// TIA Portal V20 export
FUNCTION_BLOCK "CallEquipment"   // FB134, LAD
TITLE = CallEquipment
// This block includes all general functions, checks and logik that is needed in the entire unit. E.g. general releases and system wide functionalities like air, pressure and power handling as well as general reaction to events.
// stored: IsIECCheckEnabled true, MemoryReserve 100, Namespace Unit1.Em0, SetENOAutomatically true
   VAR_INPUT
      ZoneOperationEnable { ExternalWritable := 'False'} : "LWONIK_typeSafetyZoneManualOperation";
      unitEnableControlInterfaces { ExternalWritable := 'False'} : "LAF_typeEnableControlInterfaces";
      commandExcute { ExternalWritable := 'False'} : Bool;
   END_VAR
   VAR_IN_OUT
      unitStatus : "LAF_typeUnitStatus";   // Current unit status o be used in this EM
      emFeedback : "LUC_typeEmFeedback";   // Feedback of the EM to the Unit
      unitAlarmDB : "LAF_typeAlarms";   // Summarized EM Alarms for the Unit
   END_VAR
   VAR
      instSequenceUnWinder { ExternalWritable := 'False'} : "Unit1.Em0.Sequence_1_UnWinder";   // EM Sequence Instance
      instUnWinderInitializedJob1 { ExternalWritable := 'False'} : "LAF_SelectJob";
      instUnWinderRunJob2 { ExternalWritable := 'False'} : "LAF_SelectJob";
      instUnWinderStopJob3 { ExternalWritable := 'False'} : "LAF_SelectJob";
      instUnWinderRewindJob4 { ExternalWritable := 'False'} : "LAF_SelectJob";
      instCmUnWinderAxisB { ExternalWritable := 'False'} : "LBC_AxisControl_TecPlcCn";
      instCmAirShaftOnOff { ExternalWritable := 'False'} : "LBC_TwoWayActuatorCn";
      instcmExpelFwdBwd { ExternalWritable := 'False'} : "LBC_TwoWayActuatorCn";
      instCmTensionCheckSensor { ExternalWritable := 'False'} : "LBC_DigitalSignalCn";
      instCmRadiusMeasureAnalogInput { ExternalWritable := 'False'} : "LBC_AnalogInputCn";
      instCmEpc { ExternalWritable := 'False'} : "LER_EPC_CON600";
      instCmRadiusMeasure { ExternalWritable := 'False'} : "LER_RadiusMeasure";
      instUnWinderAxisControlInterlockSummary { ExternalWritable := 'False'} : "LER_AxisControl_InterlockSummary";
      instServoTorqueCal_DR1 { ExternalWritable := 'False'} : "LER_ServoTorqueCal";
      instLDrv701ControlUnWinderAxisB { ExternalWritable := 'False'} : "LDrvSafe_SinaTlg701Control";   // Drive Telegram Function Library
      instLDrv701StatusUnWinderAxisB { ExternalWritable := 'False'} : "LDrvSafe_SinaTlg701Status";   // Drive Telegram Function Library
      statUnitStatus { ExternalWritable := 'False'} : "LAF_typeUnitStatus";   // Unit Status that is used in this project
      statAllBrakeTest { ExternalWritable := 'False'} : "LER_typeBrakeTestUnitCommands";
      instManageAlarms { ExternalWritable := 'False'} : "LAF_ManageAlarms";
      instEventsPFE { S7_SetPoint := 'True'} : "Unit1.Em0.EventsPFE";
      statEnableManualCmds { ExternalWritable := 'False'} : Bool;
      statRcEnableCmds { ExternalWritable := 'False'} : Bool;
      statPulse { ExternalWritable := 'False'} : Array[0..99] of Bool;
      statTonTimer { ExternalWritable := 'False'} : Array[0..99] of TON_TIME;
      statTofTimer { ExternalWritable := 'False'} : Array[0..99] of TOF_TIME;
      statRadius { ExternalWritable := 'False'} : LReal;
      statDiameter { ExternalWritable := 'False'} : LReal;
      citi_Ptrig : Array[0..20] of Bool;
      citiTon : Array[0..20] of TON_TIME;
      citi : Time;
      citiTest : Array[0..20] of Bool;
      SpeedLimitByRadius_Instance { S7_SetPoint := 'True'} : "Unit1.Em0.SpeedLimitByRadius";
      SpeedLimit : LReal;
      SpeedRef : LReal;
      SinaParaS_Instance { S7_SetPoint := 'True'} : SinaParaS;
   END_VAR
   VAR_TEMP
      tempScInProduction : Bool;   // Mode Production and StateComplete
      tempScNoProduction : Bool;   // Mode Manual and StateComplete
   END_VAR
   VAR CONSTANT
      TO_DO_INSERT_PRECONDITIONS_HERE : Bool := TRUE;   // Template : Add em specific conditions here
      NO_JOB : DInt;   // No job
      TRUE : Bool := TRUE;
      FALSE : Bool := FALSE;
   END_VAR
   VAR_TEMP   // added for the SCL form of the ladder/FBD networks
      _w1 : Bool;
      _w2 : Bool;
      _w3 : Bool;
      _w4 : Bool;
      _w5 : Bool;
      _w6 : Bool;
      _w7 : Bool;
      _w8 : Bool;
      _w9 : Bool;
      _w10 : Bool;
      _w11 : Bool;
      _w12 : Bool;
      _w13 : Bool;
      _w14 : Bool;
      _w15 : Bool;
   END_VAR
BEGIN

REGION Network 1: BLOCK INFO HEADER
   // (company) / (C) Copyright (year)
   // ---------------------------------------------------------------------------------
   // Title:                             (Title of this block)
   // Comment/Function: (that is implemented in the block)
   // Library/Family:           (that the source is dedicated to)
   // Author:                        (department / person in charge / contact)
   // Target System:          (test system with FW version)
   // Engineering:              TIA Portal (SW version)
   // Restrictions:               (OB types, etc.)
   // Requirements:           (hardware, technological package, etc.)
   // ---------------------------------------------------------------------------------
   // Change log table:
   // Version          | Date             | Signature      | Expert in charge  | Changes applied ------------------------|----------------------|-------------------------|--------------------------------|-----------------------
   // 001.000.000 | yyyy-mm-dd | 0x00000000 | (name of expert) | First released version
END_REGION

REGION Network 2: DESCRIPTION
   // This is a template block provided by the Automation Framework. It can be used to create an own project.
   // The Block Info Header is prepared to put in your own data.
   // Description of the block could be added here and the docu created by Code2Docu.
END_REGION

REGION Network 3: ******************** Unit Input ********************
END_REGION

REGION Network 4: Em Nodes Brake Test
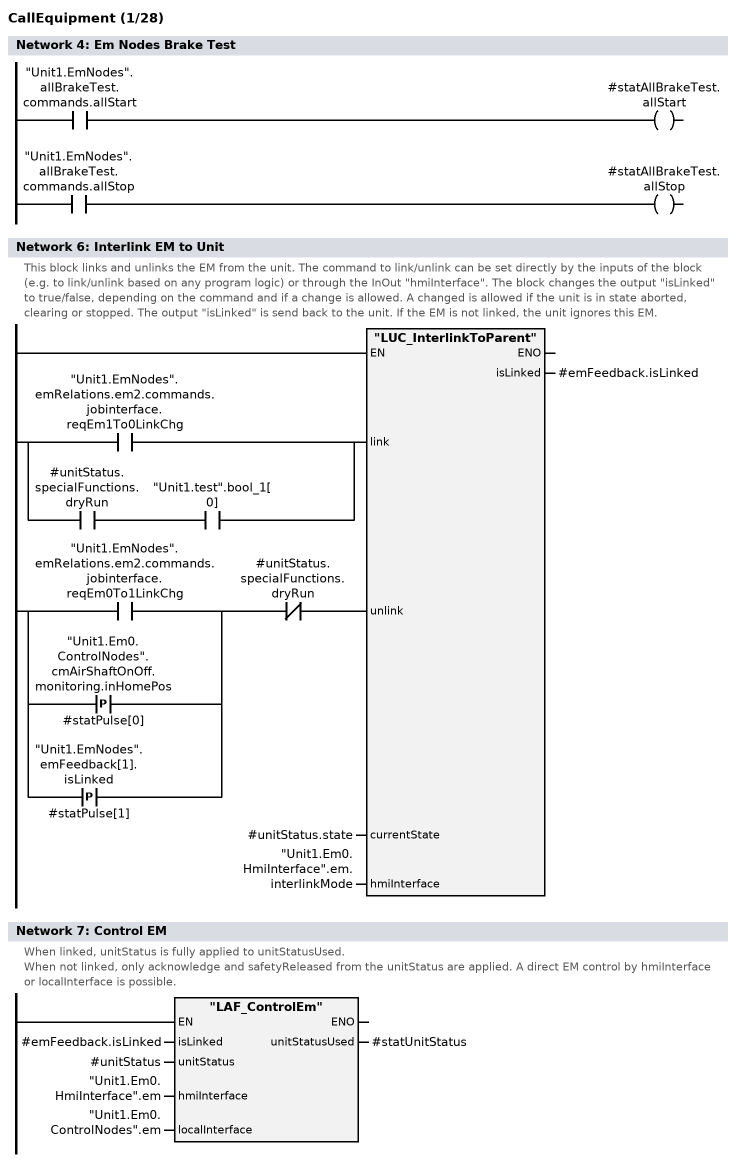
   RUNG wire#powerrail
      Contact( "Unit1.EmNodes".allBrakeTest.commands.allStart )
      Coil( #statAllBrakeTest.allStart )
   END_RUNG
   RUNG wire#powerrail
      Contact( "Unit1.EmNodes".allBrakeTest.commands.allStop )
      Coil( #statAllBrakeTest.allStop )
   END_RUNG
   // the same network as SCL:
   #statAllBrakeTest.allStart := "Unit1.EmNodes".allBrakeTest.commands.allStart;
   #statAllBrakeTest.allStop := "Unit1.EmNodes".allBrakeTest.commands.allStop;
END_REGION

REGION Network 5: ******************** Equipment Control ********************
END_REGION

REGION Network 6: Interlink EM to Unit
   // This block links and unlinks the EM from the unit. The command to link/unlink can be set directly by the inputs of the block (e.g. to link/unlink based on any program logic) or through the InOut "hmiInterface". The block changes the output "isLinked" to true/false, depending on the command and if a change is allowed. A changed is allowed if the unit is in state aborted, clearing or stopped. The output "isLinked" is send back to the unit. If the EM is not linked, the unit ignores this EM.
   RUNG wire#powerrail
      "LUC_InterlinkToParent"(link := wire#w1, unlink := wire#w3, currentState := #unitStatus.state, hmiInterface := "Unit1.Em0.HmiInterface".em.interlinkMode, isLinked => #emFeedback.isLinked)
   END_RUNG
   RUNG wire#powerrail
      Contact( "Unit1.EmNodes".emRelations.em2.commands.jobinterface.reqEm1To0LinkChg )
   END_RUNG wire#w1
   RUNG wire#powerrail
      Contact( #unitStatus.specialFunctions.dryRun )
      Contact( "Unit1.test".bool_1[0] )
   END_RUNG wire#w1
   RUNG wire#powerrail
      Contact( "Unit1.EmNodes".emRelations.em2.commands.jobinterface.reqEm0To1LinkChg )
      wire#w2
      I_Contact( #unitStatus.specialFunctions.dryRun )
   END_RUNG wire#w3
   RUNG wire#powerrail
      P_Contact(operand := "Unit1.Em0.ControlNodes".cmAirShaftOnOff.monitoring.inHomePos, bit := #statPulse[0])
   END_RUNG wire#w2
   RUNG wire#powerrail
      P_Contact(operand := "Unit1.EmNodes".emFeedback[1].isLinked, bit := #statPulse[1])
   END_RUNG wire#w2
   // the same network as SCL:
   #_w1 := "Unit1.Em0.ControlNodes".cmAirShaftOnOff.monitoring.inHomePos AND NOT #statPulse[0];   // rising edge of "Unit1.Em0.ControlNodes".cmAirShaftOnOff.monitoring.inHomePos
   #statPulse[0] := "Unit1.Em0.ControlNodes".cmAirShaftOnOff.monitoring.inHomePos;
   #_w2 := "Unit1.EmNodes".emFeedback[1].isLinked AND NOT #statPulse[1];   // rising edge of "Unit1.EmNodes".emFeedback[1].isLinked
   #statPulse[1] := "Unit1.EmNodes".emFeedback[1].isLinked;
   "LUC_InterlinkToParent"(link := "Unit1.EmNodes".emRelations.em2.commands.jobinterface.reqEm1To0LinkChg OR (#unitStatus.specialFunctions.dryRun AND "Unit1.test".bool_1[0]),
                           unlink := ("Unit1.EmNodes".emRelations.em2.commands.jobinterface.reqEm0To1LinkChg OR #_w1 OR #_w2) AND NOT #unitStatus.specialFunctions.dryRun,
                           currentState := #unitStatus.state,
                           hmiInterface := "Unit1.Em0.HmiInterface".em.interlinkMode,
                           isLinked => #emFeedback.isLinked);
END_REGION

REGION Network 7: Control EM
   // When linked, unitStatus is fully applied to unitStatusUsed.
   // When not linked, only acknowledge and safetyReleased from the unitStatus are applied. A direct EM control by hmiInterface or localInterface is possible.
   RUNG wire#powerrail
      "LAF_ControlEm"(isLinked := #emFeedback.isLinked, unitStatus := #unitStatus, hmiInterface := "Unit1.Em0.HmiInterface".em, localInterface := "Unit1.Em0.ControlNodes".em, unitStatusUsed => #statUnitStatus)
   END_RUNG
   // the same network as SCL:
   "LAF_ControlEm"(isLinked := #emFeedback.isLinked,
                   unitStatus := #unitStatus,
                   hmiInterface := "Unit1.Em0.HmiInterface".em,
                   localInterface := "Unit1.Em0.ControlNodes".em,
                   unitStatusUsed => #statUnitStatus);
END_REGION

REGION Network 8: EnableManualCmds
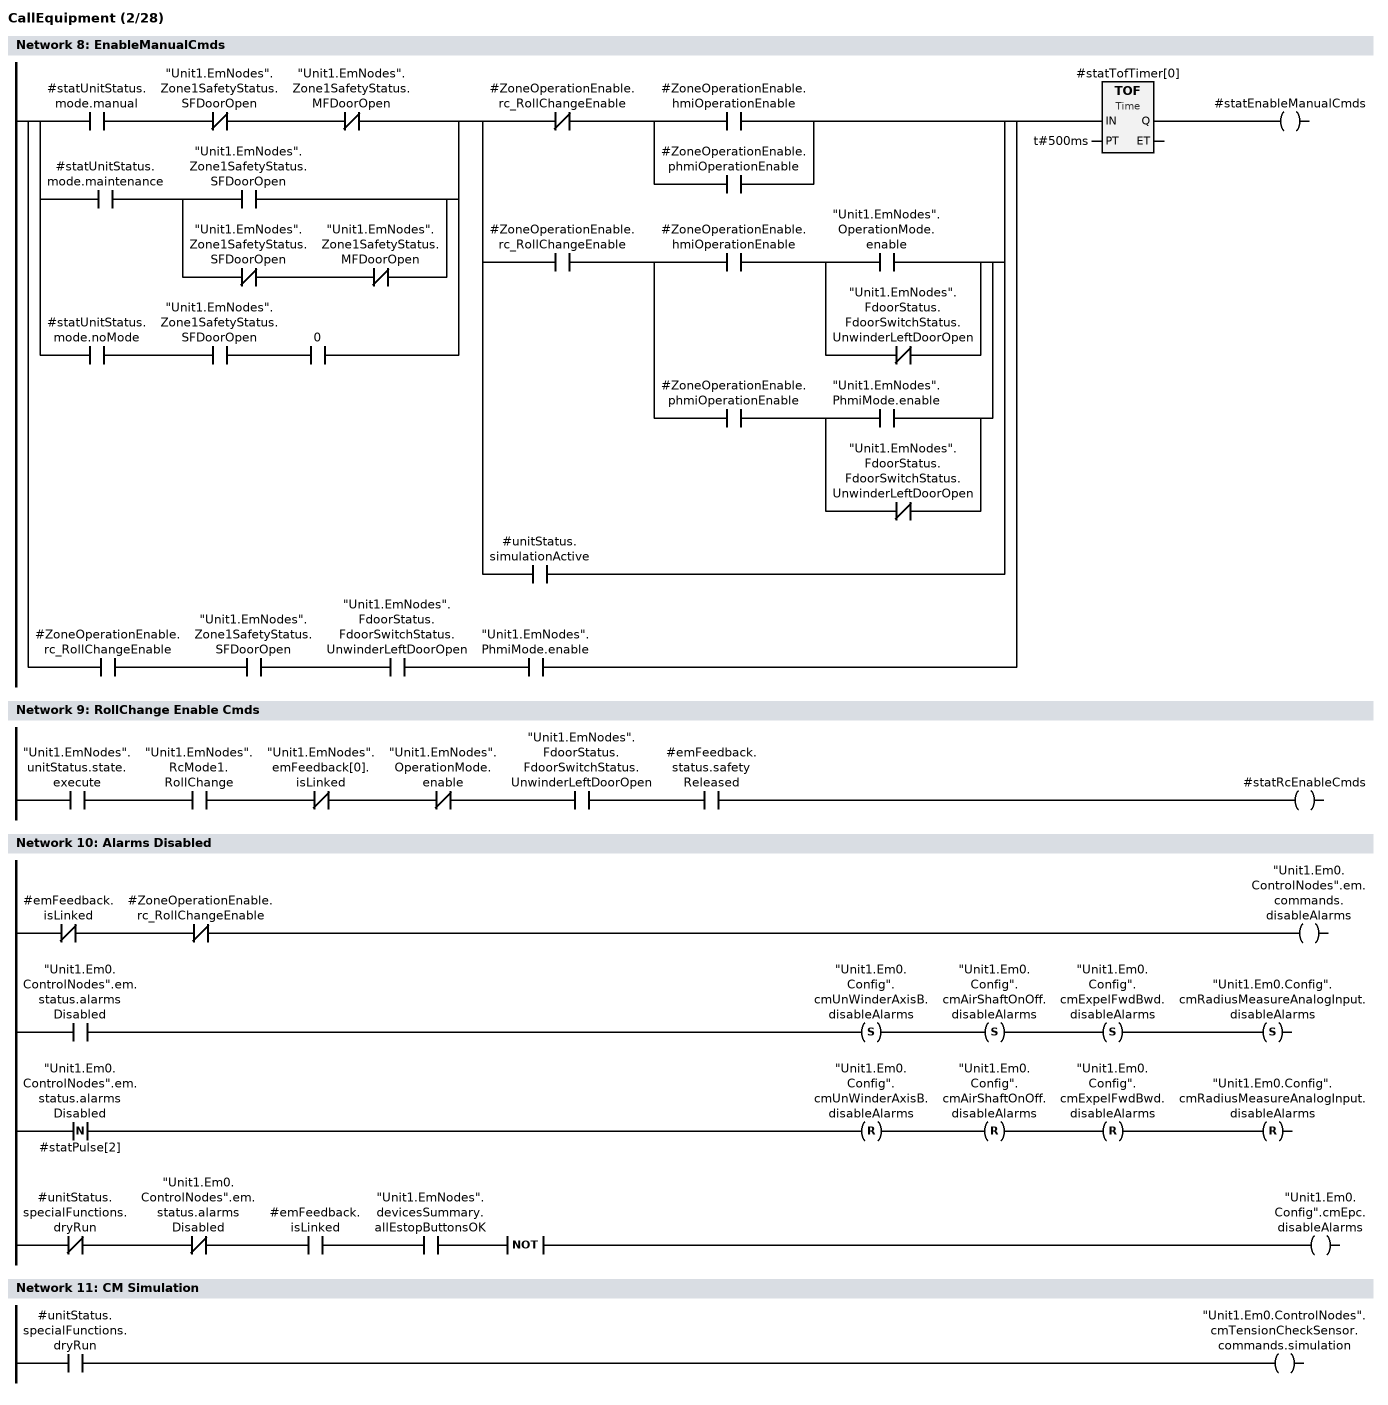
   RUNG wire#powerrail
      Contact( #statUnitStatus.mode.manual )
      I_Contact( "Unit1.EmNodes".Zone1SafetyStatus.SFDoorOpen )
      I_Contact( "Unit1.EmNodes".Zone1SafetyStatus.MFDoorOpen )
      wire#w1
      I_Contact( #ZoneOperationEnable.rc_RollChangeEnable )
      wire#w3
      Contact( #ZoneOperationEnable.hmiOperationEnable )
      wire#w4
      { S7_Templates := "time_type := Time" } #statTofTimer[0].TOF(pt := t#500ms, et =>)
      Coil( #statEnableManualCmds )
   END_RUNG
   RUNG wire#powerrail
      Contact( #statUnitStatus.mode.maintenance )
      wire#w2
      Contact( "Unit1.EmNodes".Zone1SafetyStatus.SFDoorOpen )
   END_RUNG wire#w1
   RUNG wire#w2
      I_Contact( "Unit1.EmNodes".Zone1SafetyStatus.SFDoorOpen )
      I_Contact( "Unit1.EmNodes".Zone1SafetyStatus.MFDoorOpen )
   END_RUNG wire#w1
   RUNG wire#powerrail
      Contact( #statUnitStatus.mode.noMode )
      Contact( "Unit1.EmNodes".Zone1SafetyStatus.SFDoorOpen )
      Contact( 0 )
   END_RUNG wire#w1
   RUNG wire#w3
      Contact( #ZoneOperationEnable.phmiOperationEnable )
   END_RUNG wire#w4
   RUNG wire#w1
      Contact( #ZoneOperationEnable.rc_RollChangeEnable )
      wire#w5
      Contact( #ZoneOperationEnable.hmiOperationEnable )
      wire#w6
      Contact( "Unit1.EmNodes".OperationMode.enable )
   END_RUNG wire#w4
   RUNG wire#w6
      I_Contact( "Unit1.EmNodes".FdoorStatus.FdoorSwitchStatus.UnwinderLeftDoorOpen )
   END_RUNG wire#w4
   RUNG wire#w5
      Contact( #ZoneOperationEnable.phmiOperationEnable )
      wire#w7
      Contact( "Unit1.EmNodes".PhmiMode.enable )
   END_RUNG wire#w4
   RUNG wire#w7
      I_Contact( "Unit1.EmNodes".FdoorStatus.FdoorSwitchStatus.UnwinderLeftDoorOpen )
   END_RUNG wire#w4
   RUNG wire#w1
      Contact( #unitStatus.simulationActive )
   END_RUNG wire#w4
   RUNG wire#powerrail
      Contact( #ZoneOperationEnable.rc_RollChangeEnable )
      Contact( "Unit1.EmNodes".Zone1SafetyStatus.SFDoorOpen )
      Contact( "Unit1.EmNodes".FdoorStatus.FdoorSwitchStatus.UnwinderLeftDoorOpen )
      Contact( "Unit1.EmNodes".PhmiMode.enable )
   END_RUNG wire#w4
   // the same network as SCL:
   #statTofTimer[0].TOF(IN := (((#statUnitStatus.mode.manual AND NOT "Unit1.EmNodes".Zone1SafetyStatus.SFDoorOpen AND NOT "Unit1.EmNodes".Zone1SafetyStatus.MFDoorOpen) OR (#statUnitStatus.mode.maintenance AND ("Unit1.EmNodes".Zone1SafetyStatus.SFDoorOpen OR (NOT "Unit1.EmNodes".Zone1SafetyStatus.SFDoorOpen AND NOT "Unit1.EmNodes".Zone1SafetyStatus.MFDoorOpen))) OR (#statUnitStatus.mode.noMode AND "Unit1.EmNodes".Zone1SafetyStatus.SFDoorOpen AND 0)) AND ((NOT #ZoneOperationEnable.rc_RollChangeEnable AND (#ZoneOperationEnable.hmiOperationEnable OR #ZoneOperationEnable.phmiOperationEnable)) OR (#ZoneOperationEnable.rc_RollChangeEnable AND ((#ZoneOperationEnable.hmiOperationEnable AND ("Unit1.EmNodes".OperationMode.enable OR NOT "Unit1.EmNodes".FdoorStatus.FdoorSwitchStatus.UnwinderLeftDoorOpen)) OR (#ZoneOperationEnable.phmiOperationEnable AND ("Unit1.EmNodes".PhmiMode.enable OR NOT "Unit1.EmNodes".FdoorStatus.FdoorSwitchStatus.UnwinderLeftDoorOpen)))) OR #unitStatus.simulationActive)) OR (#ZoneOperationEnable.rc_RollChangeEnable AND "Unit1.EmNodes".Zone1SafetyStatus.SFDoorOpen AND "Unit1.EmNodes".FdoorStatus.FdoorSwitchStatus.UnwinderLeftDoorOpen AND "Unit1.EmNodes".PhmiMode.enable),
                        PT := t#500ms);
   #statEnableManualCmds := #statTofTimer[0].Q;
END_REGION

REGION Network 9: RollChange Enable Cmds
   RUNG wire#powerrail
      Contact( "Unit1.EmNodes".unitStatus.state.execute )
      Contact( "Unit1.EmNodes".RcMode1.RollChange )
      I_Contact( "Unit1.EmNodes".emFeedback[0].isLinked )
      I_Contact( "Unit1.EmNodes".OperationMode.enable )
      Contact( "Unit1.EmNodes".FdoorStatus.FdoorSwitchStatus.UnwinderLeftDoorOpen )
      Contact( #emFeedback.status.safetyReleased )
      Coil( #statRcEnableCmds )
   END_RUNG
   // the same network as SCL:
   #statRcEnableCmds := "Unit1.EmNodes".unitStatus.state.execute AND "Unit1.EmNodes".RcMode1.RollChange AND NOT "Unit1.EmNodes".emFeedback[0].isLinked AND NOT "Unit1.EmNodes".OperationMode.enable AND "Unit1.EmNodes".FdoorStatus.FdoorSwitchStatus.UnwinderLeftDoorOpen AND #emFeedback.status.safetyReleased;
END_REGION

REGION Network 10: Alarms Disabled
   RUNG wire#powerrail
      I_Contact( #emFeedback.isLinked )
      I_Contact( #ZoneOperationEnable.rc_RollChangeEnable )
      Coil( "Unit1.Em0.ControlNodes".em.commands.disableAlarms )
   END_RUNG
   RUNG wire#powerrail
      Contact( "Unit1.Em0.ControlNodes".em.status.alarmsDisabled )
      S_Coil( "Unit1.Em0.Config".cmUnWinderAxisB.disableAlarms )
      S_Coil( "Unit1.Em0.Config".cmAirShaftOnOff.disableAlarms )
      S_Coil( "Unit1.Em0.Config".cmExpelFwdBwd.disableAlarms )
      S_Coil( "Unit1.Em0.Config".cmRadiusMeasureAnalogInput.disableAlarms )
   END_RUNG
   RUNG wire#powerrail
      N_Contact(operand := "Unit1.Em0.ControlNodes".em.status.alarmsDisabled, bit := #statPulse[2])
      R_Coil( "Unit1.Em0.Config".cmUnWinderAxisB.disableAlarms )
      R_Coil( "Unit1.Em0.Config".cmAirShaftOnOff.disableAlarms )
      R_Coil( "Unit1.Em0.Config".cmExpelFwdBwd.disableAlarms )
      R_Coil( "Unit1.Em0.Config".cmRadiusMeasureAnalogInput.disableAlarms )
   END_RUNG
   RUNG wire#powerrail
      I_Contact( #unitStatus.specialFunctions.dryRun )
      I_Contact( "Unit1.Em0.ControlNodes".em.status.alarmsDisabled )
      Contact( #emFeedback.isLinked )
      Contact( "Unit1.EmNodes".devicesSummary.allEstopButtonsOK )
      Not()
      Coil( "Unit1.Em0.Config".cmEpc.disableAlarms )
   END_RUNG
   // the same network as SCL:
   "Unit1.Em0.ControlNodes".em.commands.disableAlarms := NOT #emFeedback.isLinked AND NOT #ZoneOperationEnable.rc_RollChangeEnable;
   IF "Unit1.Em0.ControlNodes".em.status.alarmsDisabled THEN
       "Unit1.Em0.Config".cmUnWinderAxisB.disableAlarms := TRUE;
       "Unit1.Em0.Config".cmAirShaftOnOff.disableAlarms := TRUE;
       "Unit1.Em0.Config".cmExpelFwdBwd.disableAlarms := TRUE;
       "Unit1.Em0.Config".cmRadiusMeasureAnalogInput.disableAlarms := TRUE;
   END_IF;
   #_w1 := NOT "Unit1.Em0.ControlNodes".em.status.alarmsDisabled AND #statPulse[2];   // falling edge of "Unit1.Em0.ControlNodes".em.status.alarmsDisabled
   #statPulse[2] := "Unit1.Em0.ControlNodes".em.status.alarmsDisabled;
   IF #_w1 THEN
       "Unit1.Em0.Config".cmUnWinderAxisB.disableAlarms := FALSE;
       "Unit1.Em0.Config".cmAirShaftOnOff.disableAlarms := FALSE;
       "Unit1.Em0.Config".cmExpelFwdBwd.disableAlarms := FALSE;
       "Unit1.Em0.Config".cmRadiusMeasureAnalogInput.disableAlarms := FALSE;
   END_IF;
   "Unit1.Em0.Config".cmEpc.disableAlarms := NOT (NOT #unitStatus.specialFunctions.dryRun AND NOT "Unit1.Em0.ControlNodes".em.status.alarmsDisabled AND #emFeedback.isLinked AND "Unit1.EmNodes".devicesSummary.allEstopButtonsOK);
END_REGION

REGION Network 11: CM Simulation
   RUNG wire#powerrail
      Contact( #unitStatus.specialFunctions.dryRun )
      Coil( "Unit1.Em0.ControlNodes".cmTensionCheckSensor.commands.simulation )
   END_RUNG
   // the same network as SCL:
   "Unit1.Em0.ControlNodes".cmTensionCheckSensor.commands.simulation := #unitStatus.specialFunctions.dryRun;
END_REGION

REGION Network 12 (SCL): ReferenceDesignator
   IF "Unit1.EmNodes".unitRecipe.processUnitNo = 2 THEN
       "Unit1.Em0.Config".cmUnWinderAxisB.referenceDesignator := WSTRING#'Left UnWinder Axis B';
       "Unit1.Em0.Config".cmAirShaftOnOff.referenceDesignator := WSTRING#'Left Air Shaft';
       "Unit1.Em0.Config".cmExpelFwdBwd.referenceDesignator := WSTRING#'Left Electrode Expel';
       "Unit1.Em0.Config".cmRadiusMeasureAnalogInput.referenceDesignator := WSTRING#'Left Radius Measure';
       "Unit1.Em0.Config".cmEpc.referenceDesignator := WSTRING#'Left Uniwnder EPC';
       "Unit1.Em0.Config".cmTensionCheckSensor.referenceDesignator := WSTRING#'DigitalSignal';
   END_IF;

   IF "Unit1.EmNodes".unitRecipe.processUnitNo = 1 THEN
       "Unit1.Em0.Config".cmUnWinderAxisB.referenceDesignator := WSTRING#'RIGHT UnWinder Axis B';
       "Unit1.Em0.Config".cmAirShaftOnOff.referenceDesignator := WSTRING#'RIGHT Air Shaft';
       "Unit1.Em0.Config".cmExpelFwdBwd.referenceDesignator := WSTRING#'RIGHT Electrode Expel';
       "Unit1.Em0.Config".cmRadiusMeasureAnalogInput.referenceDesignator := WSTRING#'RIGHT Radius Measure';
       "Unit1.Em0.Config".cmEpc.referenceDesignator := WSTRING#'RIGHT Uniwnder EPC';
       "Unit1.Em0.Config".cmTensionCheckSensor.referenceDesignator := WSTRING#'DigitalSignal';
   END_IF;
END_REGION

REGION Network 13: ******************** Control Modules (Sensors) ********************
   // Call control modules that are sensors before the em logic (jobs and sequence), so that the latest value is used in the logic.
END_REGION

REGION Network 14: Reset CMS
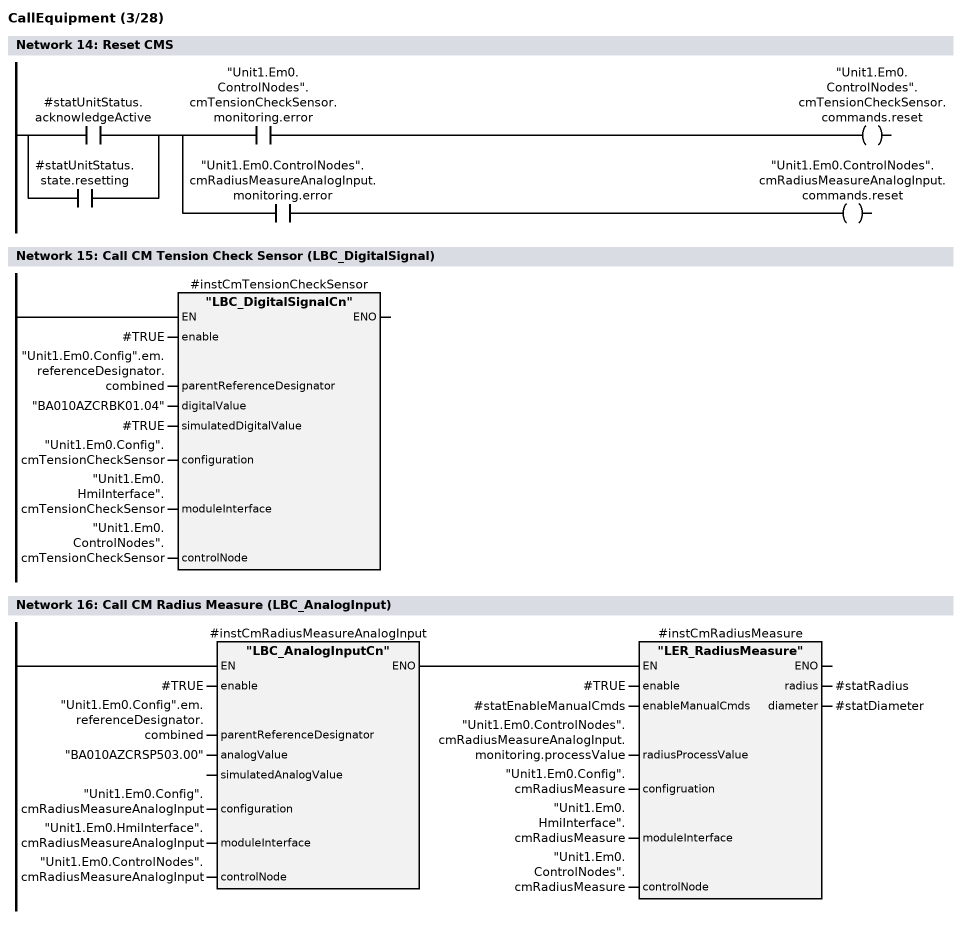
   RUNG wire#powerrail
      Contact( #statUnitStatus.acknowledgeActive )
      wire#w1
      Contact( "Unit1.Em0.ControlNodes".cmTensionCheckSensor.monitoring.error )
      Coil( "Unit1.Em0.ControlNodes".cmTensionCheckSensor.commands.reset )
   END_RUNG
   RUNG wire#powerrail
      Contact( #statUnitStatus.state.resetting )
   END_RUNG wire#w1
   RUNG wire#w1
      Contact( "Unit1.Em0.ControlNodes".cmRadiusMeasureAnalogInput.monitoring.error )
      Coil( "Unit1.Em0.ControlNodes".cmRadiusMeasureAnalogInput.commands.reset )
   END_RUNG
   // the same network as SCL:
   #_w1 := #statUnitStatus.acknowledgeActive OR #statUnitStatus.state.resetting;
   "Unit1.Em0.ControlNodes".cmTensionCheckSensor.commands.reset := #_w1 AND "Unit1.Em0.ControlNodes".cmTensionCheckSensor.monitoring.error;
   "Unit1.Em0.ControlNodes".cmRadiusMeasureAnalogInput.commands.reset := #_w1 AND "Unit1.Em0.ControlNodes".cmRadiusMeasureAnalogInput.monitoring.error;
END_REGION

REGION Network 15: Call CM Tension Check Sensor (LBC_DigitalSignal)
   RUNG wire#powerrail
      #instCmTensionCheckSensor(enable := #TRUE, parentReferenceDesignator := "Unit1.Em0.Config".em.referenceDesignator.combined, digitalValue := "BA010AZCRBK01.04", simulatedDigitalValue := #TRUE, configuration := "Unit1.Em0.Config".cmTensionCheckSensor, moduleInterface := "Unit1.Em0.HmiInterface".cmTensionCheckSensor, controlNode := "Unit1.Em0.ControlNodes".cmTensionCheckSensor)
   END_RUNG
   // the same network as SCL:
   #instCmTensionCheckSensor(enable := #TRUE,   // "LBC_DigitalSignalCn"
                           parentReferenceDesignator := "Unit1.Em0.Config".em.referenceDesignator.combined,
                           digitalValue := "BA010AZCRBK01.04",
                           simulatedDigitalValue := #TRUE,
                           configuration := "Unit1.Em0.Config".cmTensionCheckSensor,
                           moduleInterface := "Unit1.Em0.HmiInterface".cmTensionCheckSensor,
                           controlNode := "Unit1.Em0.ControlNodes".cmTensionCheckSensor);
END_REGION

REGION Network 16: Call CM Radius Measure (LBC_AnalogInput)
   RUNG wire#powerrail
      #instCmRadiusMeasureAnalogInput(enable := #TRUE, parentReferenceDesignator := "Unit1.Em0.Config".em.referenceDesignator.combined, analogValue := "BA010AZCRSP503.00", simulatedAnalogValue :=, configuration := "Unit1.Em0.Config".cmRadiusMeasureAnalogInput, moduleInterface := "Unit1.Em0.HmiInterface".cmRadiusMeasureAnalogInput, controlNode := "Unit1.Em0.ControlNodes".cmRadiusMeasureAnalogInput)
      #instCmRadiusMeasure(enable := #TRUE, enableManualCmds := #statEnableManualCmds, radiusProcessValue := "Unit1.Em0.ControlNodes".cmRadiusMeasureAnalogInput.monitoring.processValue, configruation := "Unit1.Em0.Config".cmRadiusMeasure, moduleInterface := "Unit1.Em0.HmiInterface".cmRadiusMeasure, controlNode := "Unit1.Em0.ControlNodes".cmRadiusMeasure, radius => #statRadius, diameter => #statDiameter)
   END_RUNG
   // the same network as SCL:
   #instCmRadiusMeasureAnalogInput(enable := #TRUE,   // "LBC_AnalogInputCn"
                           parentReferenceDesignator := "Unit1.Em0.Config".em.referenceDesignator.combined,
                           analogValue := "BA010AZCRSP503.00",
                           configuration := "Unit1.Em0.Config".cmRadiusMeasureAnalogInput,
                           moduleInterface := "Unit1.Em0.HmiInterface".cmRadiusMeasureAnalogInput,
                           controlNode := "Unit1.Em0.ControlNodes".cmRadiusMeasureAnalogInput,
                           ENO => #_w1);
   IF #_w1 THEN
       #instCmRadiusMeasure(enable := #TRUE,   // "LER_RadiusMeasure"
                            enableManualCmds := #statEnableManualCmds,
                            radiusProcessValue := "Unit1.Em0.ControlNodes".cmRadiusMeasureAnalogInput.monitoring.processValue,
                            configruation := "Unit1.Em0.Config".cmRadiusMeasure,
                            moduleInterface := "Unit1.Em0.HmiInterface".cmRadiusMeasure,
                            controlNode := "Unit1.Em0.ControlNodes".cmRadiusMeasure,
                            radius => #statRadius,
                            diameter => #statDiameter);
   END_IF;
END_REGION

REGION Network 17: ******************** Equipment Logic ********************
END_REGION

REGION Network 18: Map Unit Status to Sequence Status [1] UnWinder
   // This block maps the unit status to the seuqnce status. Thus, it controls the sequence depending on the unit status. E.g. it sets the sequence to automatic when the unit state is in productions. This blocks work perfectly with the sequences provided in the AF. 
   // This typed block (MapUnitStatusToSequence) could be adjusted to specific application requirements or if other, user-defined sequences are used.
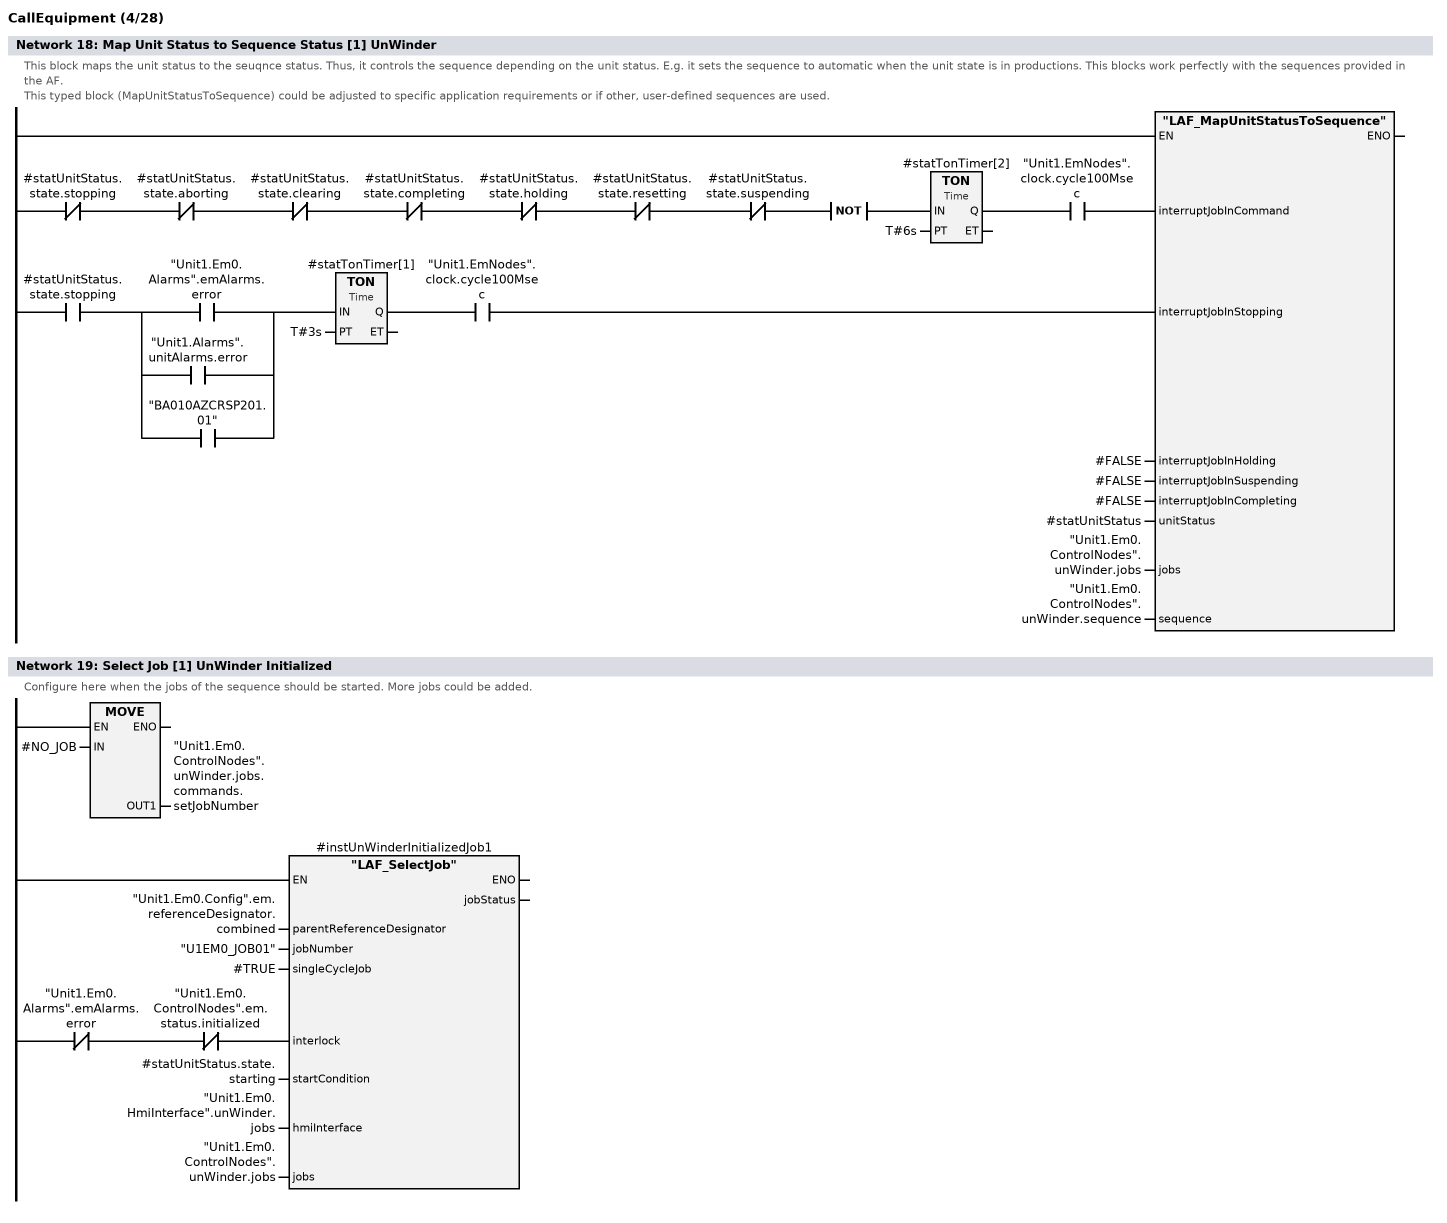
   RUNG wire#powerrail
      "LAF_MapUnitStatusToSequence"(interruptJobInCommand := wire#w1, interruptJobInStopping := wire#w4, interruptJobInHolding := #FALSE, interruptJobInSuspending := #FALSE, interruptJobInCompleting := #FALSE, unitStatus := #statUnitStatus, jobs := "Unit1.Em0.ControlNodes".unWinder.jobs, sequence := "Unit1.Em0.ControlNodes".unWinder.sequence)
   END_RUNG
   RUNG wire#powerrail
      I_Contact( #statUnitStatus.state.stopping )
      I_Contact( #statUnitStatus.state.aborting )
      I_Contact( #statUnitStatus.state.clearing )
      I_Contact( #statUnitStatus.state.completing )
      I_Contact( #statUnitStatus.state.holding )
      I_Contact( #statUnitStatus.state.resetting )
      I_Contact( #statUnitStatus.state.suspending )
      Not()
      { S7_Templates := "time_type := Time" } #statTonTimer[2].TON(pt := T#6s, et =>)
      Contact( "Unit1.EmNodes".clock.cycle100Msec )
   END_RUNG wire#w1
   RUNG wire#powerrail
      Contact( #statUnitStatus.state.stopping )
      wire#w2
      Contact( "Unit1.Em0.Alarms".emAlarms.error )
      wire#w3
      { S7_Templates := "time_type := Time" } #statTonTimer[1].TON(pt := T#3s, et =>)
      Contact( "Unit1.EmNodes".clock.cycle100Msec )
   END_RUNG wire#w4
   RUNG wire#w2
      Contact( "Unit1.Alarms".unitAlarms.error )
   END_RUNG wire#w3
   RUNG wire#w2
      Contact( "BA010AZCRSP201.01" )
   END_RUNG wire#w3
   // the same network as SCL:
   #statTonTimer[2].TON(IN := NOT (NOT #statUnitStatus.state.stopping AND NOT #statUnitStatus.state.aborting AND NOT #statUnitStatus.state.clearing AND NOT #statUnitStatus.state.completing AND NOT #statUnitStatus.state.holding AND NOT #statUnitStatus.state.resetting AND NOT #statUnitStatus.state.suspending),
                        PT := T#6s);
   #_w1 := #statTonTimer[2].Q AND "Unit1.EmNodes".clock.cycle100Msec;
   #statTonTimer[1].TON(IN := #statUnitStatus.state.stopping AND ("Unit1.Em0.Alarms".emAlarms.error OR "Unit1.Alarms".unitAlarms.error OR "BA010AZCRSP201.01"),
                        PT := T#3s);
   "LAF_MapUnitStatusToSequence"(interruptJobInCommand := #_w1,
                           interruptJobInStopping := #statTonTimer[1].Q AND "Unit1.EmNodes".clock.cycle100Msec,
                           interruptJobInHolding := #FALSE,
                           interruptJobInSuspending := #FALSE,
                           interruptJobInCompleting := #FALSE,
                           unitStatus := #statUnitStatus,
                           jobs := "Unit1.Em0.ControlNodes".unWinder.jobs,
                           sequence := "Unit1.Em0.ControlNodes".unWinder.sequence);
END_REGION

REGION Network 19: Select Job [1] UnWinder Initialized
   // Configure here when the jobs of the sequence should be started. More jobs could be added.
   RUNG wire#powerrail
      Move(in := #NO_JOB, out1 => "Unit1.Em0.ControlNodes".unWinder.jobs.commands.setJobNumber)
   END_RUNG
   RUNG wire#powerrail
      #instUnWinderInitializedJob1(interlock := wire#w1, parentReferenceDesignator := "Unit1.Em0.Config".em.referenceDesignator.combined, jobNumber := "U1EM0_JOB01", singleCycleJob := #TRUE, startCondition := #statUnitStatus.state.starting, hmiInterface := "Unit1.Em0.HmiInterface".unWinder.jobs, jobs := "Unit1.Em0.ControlNodes".unWinder.jobs, jobStatus =>)
   END_RUNG
   RUNG wire#powerrail
      I_Contact( "Unit1.Em0.Alarms".emAlarms.error )
      I_Contact( "Unit1.Em0.ControlNodes".em.status.initialized )
   END_RUNG wire#w1
   // the same network as SCL:
   "Unit1.Em0.ControlNodes".unWinder.jobs.commands.setJobNumber := #NO_JOB;
   #instUnWinderInitializedJob1(parentReferenceDesignator := "Unit1.Em0.Config".em.referenceDesignator.combined,   // "LAF_SelectJob"
                           jobNumber := "U1EM0_JOB01",
                           singleCycleJob := #TRUE,
                           interlock := NOT "Unit1.Em0.Alarms".emAlarms.error AND NOT "Unit1.Em0.ControlNodes".em.status.initialized,
                           startCondition := #statUnitStatus.state.starting,
                           hmiInterface := "Unit1.Em0.HmiInterface".unWinder.jobs,
                           jobs := "Unit1.Em0.ControlNodes".unWinder.jobs);
END_REGION

REGION Network 20: Select Job [2] UnWinder Run
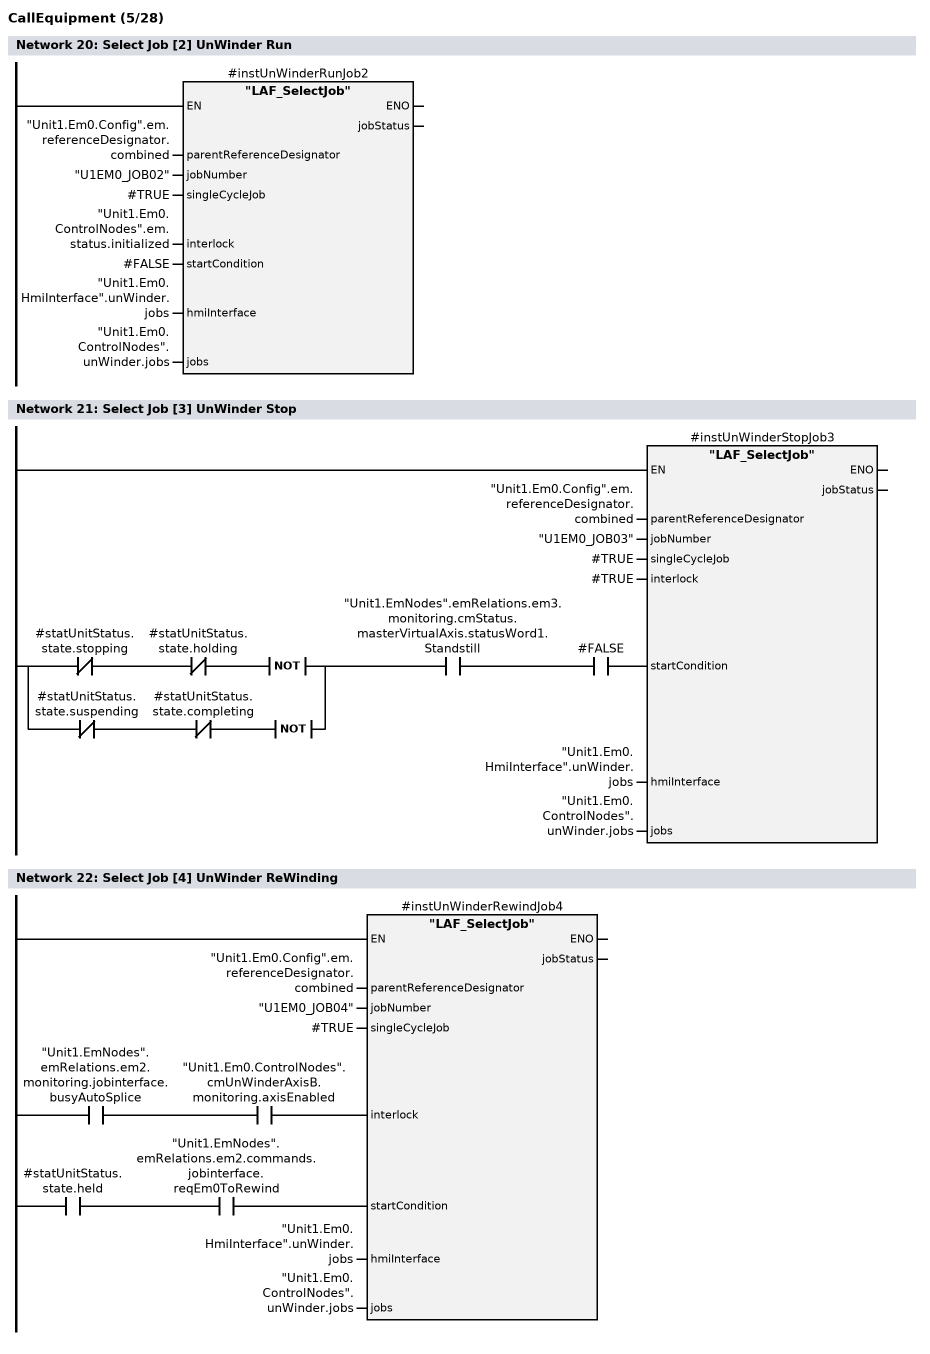
   RUNG wire#powerrail
      #instUnWinderRunJob2(parentReferenceDesignator := "Unit1.Em0.Config".em.referenceDesignator.combined, jobNumber := "U1EM0_JOB02", singleCycleJob := #TRUE, interlock := "Unit1.Em0.ControlNodes".em.status.initialized, startCondition := #FALSE, hmiInterface := "Unit1.Em0.HmiInterface".unWinder.jobs, jobs := "Unit1.Em0.ControlNodes".unWinder.jobs, jobStatus =>)
   END_RUNG
   // the same network as SCL:
   #instUnWinderRunJob2(parentReferenceDesignator := "Unit1.Em0.Config".em.referenceDesignator.combined,   // "LAF_SelectJob"
                        jobNumber := "U1EM0_JOB02",
                        singleCycleJob := #TRUE,
                        interlock := "Unit1.Em0.ControlNodes".em.status.initialized,
                        startCondition := #FALSE,
                        hmiInterface := "Unit1.Em0.HmiInterface".unWinder.jobs,
                        jobs := "Unit1.Em0.ControlNodes".unWinder.jobs);
END_REGION

REGION Network 21: Select Job [3] UnWinder Stop
   RUNG wire#powerrail
      #instUnWinderStopJob3(startCondition := wire#w2, parentReferenceDesignator := "Unit1.Em0.Config".em.referenceDesignator.combined, jobNumber := "U1EM0_JOB03", singleCycleJob := #TRUE, interlock := #TRUE, hmiInterface := "Unit1.Em0.HmiInterface".unWinder.jobs, jobs := "Unit1.Em0.ControlNodes".unWinder.jobs, jobStatus =>)
   END_RUNG
   RUNG wire#powerrail
      I_Contact( #statUnitStatus.state.stopping )
      I_Contact( #statUnitStatus.state.holding )
      Not()
      wire#w1
      Contact( "Unit1.EmNodes".emRelations.em3.monitoring.cmStatus.masterVirtualAxis.statusWord1.Standstill )
      Contact( #FALSE )
   END_RUNG wire#w2
   RUNG wire#powerrail
      I_Contact( #statUnitStatus.state.suspending )
      I_Contact( #statUnitStatus.state.completing )
      Not()
   END_RUNG wire#w1
   // the same network as SCL:
   #instUnWinderStopJob3(parentReferenceDesignator := "Unit1.Em0.Config".em.referenceDesignator.combined,   // "LAF_SelectJob"
                         jobNumber := "U1EM0_JOB03",
                         singleCycleJob := #TRUE,
                         interlock := #TRUE,
                         startCondition := (NOT (NOT #statUnitStatus.state.stopping AND NOT #statUnitStatus.state.holding) OR NOT (NOT #statUnitStatus.state.suspending AND NOT #statUnitStatus.state.completing)) AND "Unit1.EmNodes".emRelations.em3.monitoring.cmStatus.masterVirtualAxis.statusWord1.Standstill AND #FALSE,
                         hmiInterface := "Unit1.Em0.HmiInterface".unWinder.jobs,
                         jobs := "Unit1.Em0.ControlNodes".unWinder.jobs);
END_REGION

REGION Network 22: Select Job [4] UnWinder ReWinding
   RUNG wire#powerrail
      #instUnWinderRewindJob4(interlock := wire#w1, startCondition := wire#w2, parentReferenceDesignator := "Unit1.Em0.Config".em.referenceDesignator.combined, jobNumber := "U1EM0_JOB04", singleCycleJob := #TRUE, hmiInterface := "Unit1.Em0.HmiInterface".unWinder.jobs, jobs := "Unit1.Em0.ControlNodes".unWinder.jobs, jobStatus =>)
   END_RUNG
   RUNG wire#powerrail
      Contact( "Unit1.EmNodes".emRelations.em2.monitoring.jobinterface.busyAutoSplice )
      Contact( "Unit1.Em0.ControlNodes".cmUnWinderAxisB.monitoring.axisEnabled )
   END_RUNG wire#w1
   RUNG wire#powerrail
      Contact( #statUnitStatus.state.held )
      Contact( "Unit1.EmNodes".emRelations.em2.commands.jobinterface.reqEm0ToRewind )
   END_RUNG wire#w2
   // the same network as SCL:
   #instUnWinderRewindJob4(parentReferenceDesignator := "Unit1.Em0.Config".em.referenceDesignator.combined,   // "LAF_SelectJob"
                           jobNumber := "U1EM0_JOB04",
                           singleCycleJob := #TRUE,
                           interlock := "Unit1.EmNodes".emRelations.em2.monitoring.jobinterface.busyAutoSplice AND "Unit1.Em0.ControlNodes".cmUnWinderAxisB.monitoring.axisEnabled,
                           startCondition := #statUnitStatus.state.held AND "Unit1.EmNodes".emRelations.em2.commands.jobinterface.reqEm0ToRewind,
                           hmiInterface := "Unit1.Em0.HmiInterface".unWinder.jobs,
                           jobs := "Unit1.Em0.ControlNodes".unWinder.jobs);
END_REGION

REGION Network 23: Select Job Working Done
END_REGION

REGION Network 24: EM Control Select Job Move
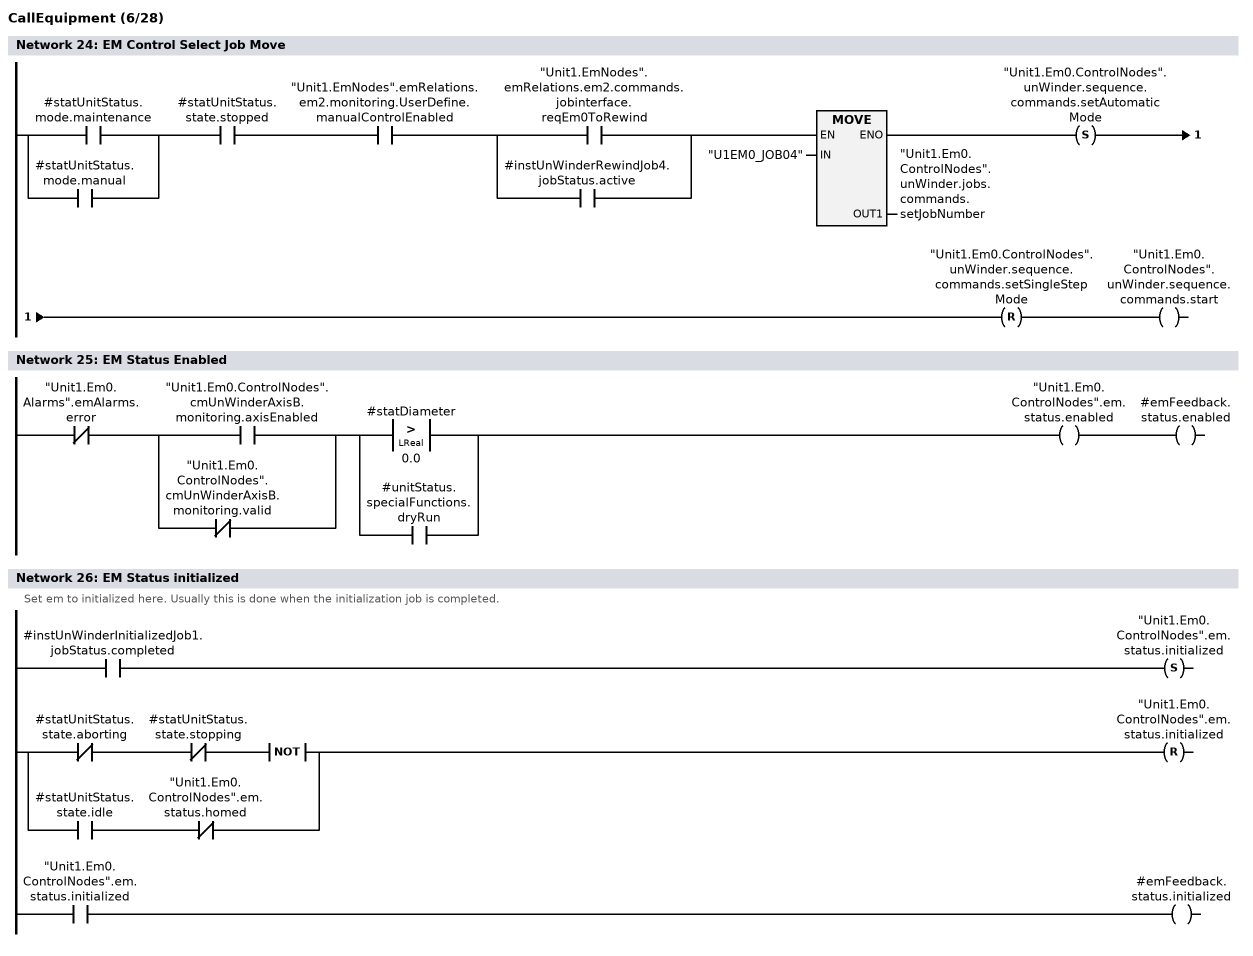
   RUNG wire#powerrail
      Contact( #statUnitStatus.mode.maintenance )
      wire#w1
      Contact( #statUnitStatus.state.stopped )
      Contact( "Unit1.EmNodes".emRelations.em2.monitoring.UserDefine.manualControlEnabled )
      wire#w2
      Contact( "Unit1.EmNodes".emRelations.em2.commands.jobinterface.reqEm0ToRewind )
      wire#w3
      Move(in := "U1EM0_JOB04", out1 => "Unit1.Em0.ControlNodes".unWinder.jobs.commands.setJobNumber)
      S_Coil( "Unit1.Em0.ControlNodes".unWinder.sequence.commands.setAutomaticMode )
      R_Coil( "Unit1.Em0.ControlNodes".unWinder.sequence.commands.setSingleStepMode )
      Coil( "Unit1.Em0.ControlNodes".unWinder.sequence.commands.start )
   END_RUNG
   RUNG wire#powerrail
      Contact( #statUnitStatus.mode.manual )
   END_RUNG wire#w1
   RUNG wire#w2
      Contact( #instUnWinderRewindJob4.jobStatus.active )
   END_RUNG wire#w3
   // the same network as SCL:
   #_w1 := (#statUnitStatus.mode.maintenance OR #statUnitStatus.mode.manual) AND #statUnitStatus.state.stopped AND "Unit1.EmNodes".emRelations.em2.monitoring.UserDefine.manualControlEnabled AND ("Unit1.EmNodes".emRelations.em2.commands.jobinterface.reqEm0ToRewind OR #instUnWinderRewindJob4.jobStatus.active);
   IF #_w1 THEN
       "Unit1.Em0.ControlNodes".unWinder.jobs.commands.setJobNumber := "U1EM0_JOB04";
       "Unit1.Em0.ControlNodes".unWinder.sequence.commands.setAutomaticMode := TRUE;
       "Unit1.Em0.ControlNodes".unWinder.sequence.commands.setSingleStepMode := FALSE;
   END_IF;
   "Unit1.Em0.ControlNodes".unWinder.sequence.commands.start := #_w1;
END_REGION

REGION Network 25: EM Status Enabled
   RUNG wire#powerrail
      I_Contact( "Unit1.Em0.Alarms".emAlarms.error )
      wire#w1
      Contact( "Unit1.Em0.ControlNodes".cmUnWinderAxisB.monitoring.axisEnabled )
      wire#w2
      { S7_Templates := "SrcType := LReal" } GT_Contact(in1 := #statDiameter, in2 := 0.0)
      wire#w3
      Coil( "Unit1.Em0.ControlNodes".em.status.enabled )
      Coil( #emFeedback.status.enabled )
   END_RUNG
   RUNG wire#w1
      I_Contact( "Unit1.Em0.ControlNodes".cmUnWinderAxisB.monitoring.valid )
   END_RUNG wire#w2
   RUNG wire#w2
      Contact( #unitStatus.specialFunctions.dryRun )
   END_RUNG wire#w3
   // the same network as SCL:
   "Unit1.Em0.ControlNodes".em.status.enabled := NOT "Unit1.Em0.Alarms".emAlarms.error AND ("Unit1.Em0.ControlNodes".cmUnWinderAxisB.monitoring.axisEnabled OR NOT "Unit1.Em0.ControlNodes".cmUnWinderAxisB.monitoring.valid) AND ((#statDiameter > 0.0) OR #unitStatus.specialFunctions.dryRun);
   #emFeedback.status.enabled := "Unit1.Em0.ControlNodes".em.status.enabled;
END_REGION

REGION Network 26: EM Status initialized
   // Set em to initialized here. Usually this is done when the initialization job is completed.
   RUNG wire#powerrail
      Contact( #instUnWinderInitializedJob1.jobStatus.completed )
      S_Coil( "Unit1.Em0.ControlNodes".em.status.initialized )
   END_RUNG
   RUNG wire#powerrail
      I_Contact( #statUnitStatus.state.aborting )
      I_Contact( #statUnitStatus.state.stopping )
      Not()
      wire#w1
      R_Coil( "Unit1.Em0.ControlNodes".em.status.initialized )
   END_RUNG
   RUNG wire#powerrail
      Contact( #statUnitStatus.state.idle )
      I_Contact( "Unit1.Em0.ControlNodes".em.status.homed )
   END_RUNG wire#w1
   RUNG wire#powerrail
      Contact( "Unit1.Em0.ControlNodes".em.status.initialized )
      Coil( #emFeedback.status.initialized )
   END_RUNG
   // the same network as SCL:
   IF #instUnWinderInitializedJob1.jobStatus.completed THEN
       "Unit1.Em0.ControlNodes".em.status.initialized := TRUE;
   END_IF;
   IF NOT (NOT #statUnitStatus.state.aborting AND NOT #statUnitStatus.state.stopping) OR (#statUnitStatus.state.idle AND NOT "Unit1.Em0.ControlNodes".em.status.homed) THEN
       "Unit1.Em0.ControlNodes".em.status.initialized := FALSE;
   END_IF;
   #emFeedback.status.initialized := "Unit1.Em0.ControlNodes".em.status.initialized;
END_REGION

REGION Network 27: EM Status Homed
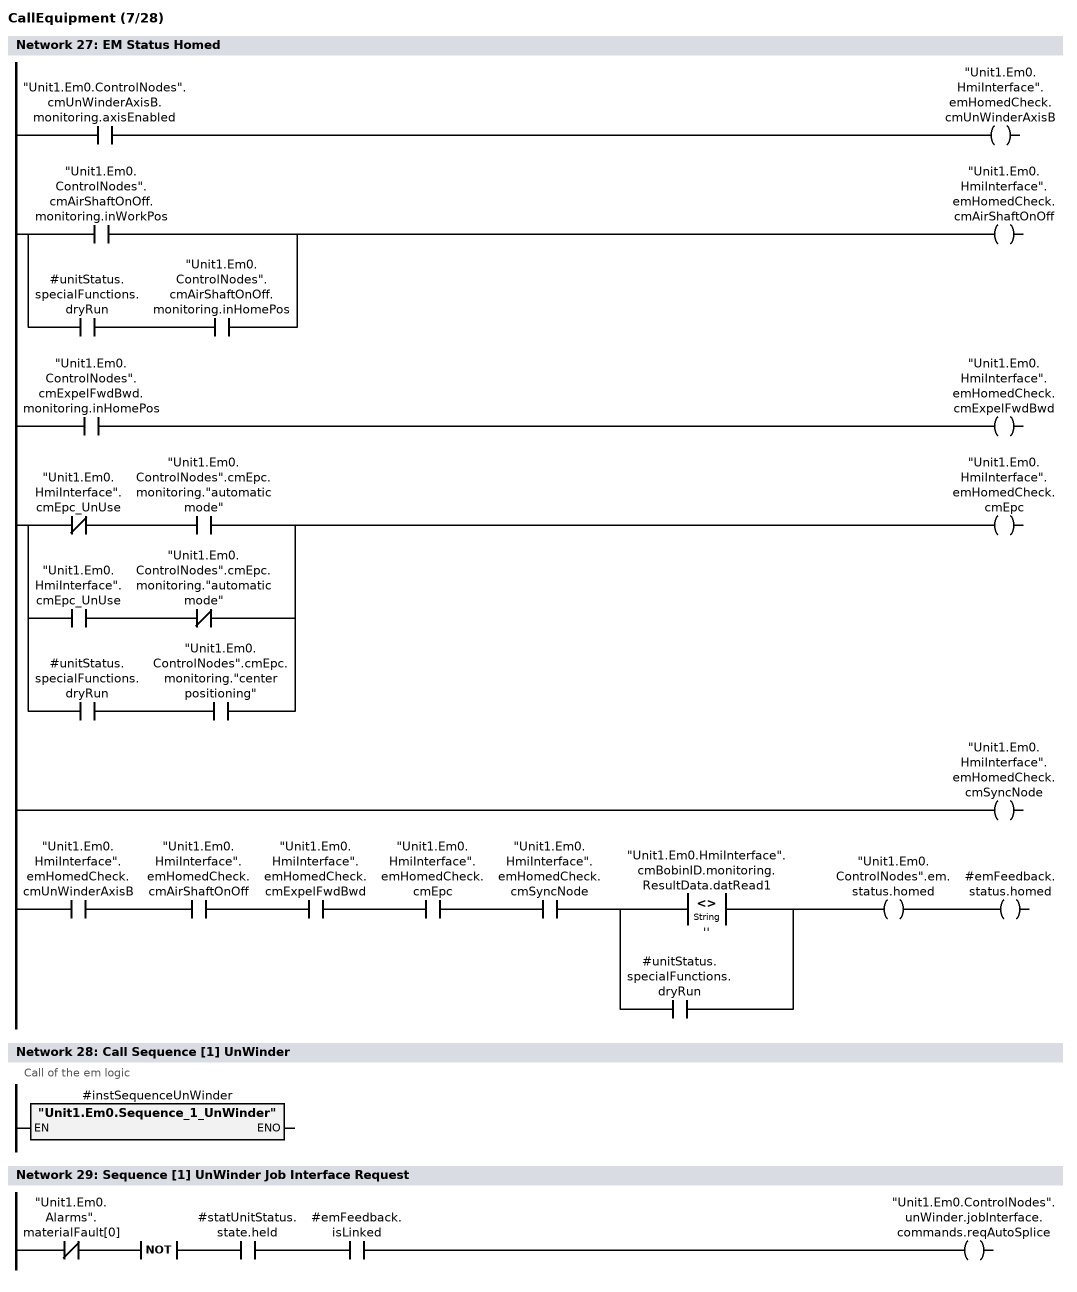
   RUNG wire#powerrail
      Contact( "Unit1.Em0.ControlNodes".cmUnWinderAxisB.monitoring.axisEnabled )
      Coil( "Unit1.Em0.HmiInterface".emHomedCheck.cmUnWinderAxisB )
   END_RUNG
   RUNG wire#powerrail
      Contact( "Unit1.Em0.ControlNodes".cmAirShaftOnOff.monitoring.inWorkPos )
      wire#w1
      Coil( "Unit1.Em0.HmiInterface".emHomedCheck.cmAirShaftOnOff )
   END_RUNG
   RUNG wire#powerrail
      Contact( #unitStatus.specialFunctions.dryRun )
      Contact( "Unit1.Em0.ControlNodes".cmAirShaftOnOff.monitoring.inHomePos )
   END_RUNG wire#w1
   RUNG wire#powerrail
      Contact( "Unit1.Em0.ControlNodes".cmExpelFwdBwd.monitoring.inHomePos )
      Coil( "Unit1.Em0.HmiInterface".emHomedCheck.cmExpelFwdBwd )
   END_RUNG
   RUNG wire#powerrail
      I_Contact( "Unit1.Em0.HmiInterface".cmEpc_UnUse )
      Contact( "Unit1.Em0.ControlNodes".cmEpc.monitoring."automatic mode" )
      wire#w2
      Coil( "Unit1.Em0.HmiInterface".emHomedCheck.cmEpc )
   END_RUNG
   RUNG wire#powerrail
      Contact( "Unit1.Em0.HmiInterface".cmEpc_UnUse )
      I_Contact( "Unit1.Em0.ControlNodes".cmEpc.monitoring."automatic mode" )
   END_RUNG wire#w2
   RUNG wire#powerrail
      Contact( #unitStatus.specialFunctions.dryRun )
      Contact( "Unit1.Em0.ControlNodes".cmEpc.monitoring."center positioning" )
   END_RUNG wire#w2
   RUNG wire#powerrail
      Coil( "Unit1.Em0.HmiInterface".emHomedCheck.cmSyncNode )
   END_RUNG
   RUNG wire#powerrail
      Contact( "Unit1.Em0.HmiInterface".emHomedCheck.cmUnWinderAxisB )
      Contact( "Unit1.Em0.HmiInterface".emHomedCheck.cmAirShaftOnOff )
      Contact( "Unit1.Em0.HmiInterface".emHomedCheck.cmExpelFwdBwd )
      Contact( "Unit1.Em0.HmiInterface".emHomedCheck.cmEpc )
      Contact( "Unit1.Em0.HmiInterface".emHomedCheck.cmSyncNode )
      wire#w3
      { S7_Templates := "SrcType := String" } NE_Contact(in1 := "Unit1.Em0.HmiInterface".cmBobinID.monitoring.ResultData.datRead1, in2 := '')
      wire#w4
      Coil( "Unit1.Em0.ControlNodes".em.status.homed )
      Coil( #emFeedback.status.homed )
   END_RUNG
   RUNG wire#w3
      Contact( #unitStatus.specialFunctions.dryRun )
   END_RUNG wire#w4
   // the same network as SCL:
   "Unit1.Em0.HmiInterface".emHomedCheck.cmUnWinderAxisB := "Unit1.Em0.ControlNodes".cmUnWinderAxisB.monitoring.axisEnabled;
   "Unit1.Em0.HmiInterface".emHomedCheck.cmAirShaftOnOff := "Unit1.Em0.ControlNodes".cmAirShaftOnOff.monitoring.inWorkPos OR (#unitStatus.specialFunctions.dryRun AND "Unit1.Em0.ControlNodes".cmAirShaftOnOff.monitoring.inHomePos);
   "Unit1.Em0.HmiInterface".emHomedCheck.cmExpelFwdBwd := "Unit1.Em0.ControlNodes".cmExpelFwdBwd.monitoring.inHomePos;
   "Unit1.Em0.HmiInterface".emHomedCheck.cmEpc := (NOT "Unit1.Em0.HmiInterface".cmEpc_UnUse AND "Unit1.Em0.ControlNodes".cmEpc.monitoring."automatic mode") OR ("Unit1.Em0.HmiInterface".cmEpc_UnUse AND NOT "Unit1.Em0.ControlNodes".cmEpc.monitoring."automatic mode") OR (#unitStatus.specialFunctions.dryRun AND "Unit1.Em0.ControlNodes".cmEpc.monitoring."center positioning");
   "Unit1.Em0.HmiInterface".emHomedCheck.cmSyncNode := TRUE;
   "Unit1.Em0.ControlNodes".em.status.homed := "Unit1.Em0.HmiInterface".emHomedCheck.cmUnWinderAxisB AND "Unit1.Em0.HmiInterface".emHomedCheck.cmAirShaftOnOff AND "Unit1.Em0.HmiInterface".emHomedCheck.cmExpelFwdBwd AND "Unit1.Em0.HmiInterface".emHomedCheck.cmEpc AND "Unit1.Em0.HmiInterface".emHomedCheck.cmSyncNode AND (("Unit1.Em0.HmiInterface".cmBobinID.monitoring.ResultData.datRead1 <> '') OR #unitStatus.specialFunctions.dryRun);
   #emFeedback.status.homed := "Unit1.Em0.ControlNodes".em.status.homed;
END_REGION

REGION Network 28: Call Sequence [1] UnWinder
   // Call of the em logic
   RUNG wire#powerrail
      #instSequenceUnWinder()
   END_RUNG
   // the same network as SCL:
   #instSequenceUnWinder();   // "Unit1.Em0.Sequence_1_UnWinder"
END_REGION

REGION Network 29: Sequence [1] UnWinder Job Interface Request
   RUNG wire#powerrail
      I_Contact( "Unit1.Em0.Alarms".materialFault[0] )
      Not()
      Contact( #statUnitStatus.state.held )
      Contact( #emFeedback.isLinked )
      Coil( "Unit1.Em0.ControlNodes".unWinder.jobInterface.commands.reqAutoSplice )
   END_RUNG
   // the same network as SCL:
   "Unit1.Em0.ControlNodes".unWinder.jobInterface.commands.reqAutoSplice := NOT (NOT "Unit1.Em0.Alarms".materialFault[0]) AND #statUnitStatus.state.held AND #emFeedback.isLinked;
END_REGION

REGION Network 30: Sequence [1] Unwinder Job Interface Busy
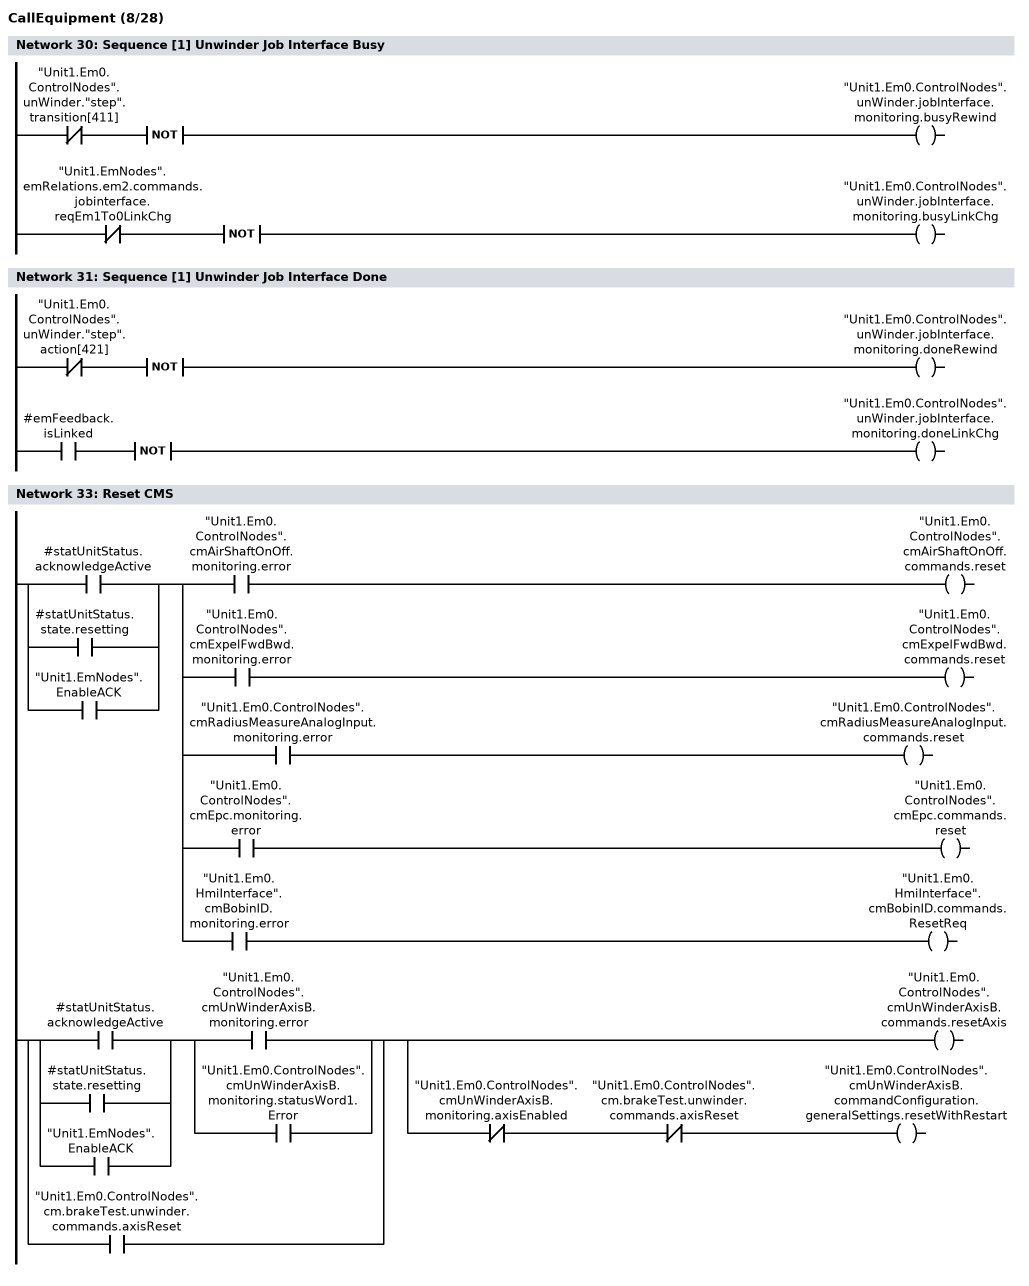
   RUNG wire#powerrail
      I_Contact( "Unit1.Em0.ControlNodes".unWinder."step".transition[411] )
      Not()
      Coil( "Unit1.Em0.ControlNodes".unWinder.jobInterface.monitoring.busyRewind )
   END_RUNG
   RUNG wire#powerrail
      I_Contact( "Unit1.EmNodes".emRelations.em2.commands.jobinterface.reqEm1To0LinkChg )
      Not()
      Coil( "Unit1.Em0.ControlNodes".unWinder.jobInterface.monitoring.busyLinkChg )
   END_RUNG
   // the same network as SCL:
   "Unit1.Em0.ControlNodes".unWinder.jobInterface.monitoring.busyRewind := NOT (NOT "Unit1.Em0.ControlNodes".unWinder."step".transition[411]);
   "Unit1.Em0.ControlNodes".unWinder.jobInterface.monitoring.busyLinkChg := NOT (NOT "Unit1.EmNodes".emRelations.em2.commands.jobinterface.reqEm1To0LinkChg);
END_REGION

REGION Network 31: Sequence [1] Unwinder Job Interface Done
   RUNG wire#powerrail
      I_Contact( "Unit1.Em0.ControlNodes".unWinder."step".action[421] )
      Not()
      Coil( "Unit1.Em0.ControlNodes".unWinder.jobInterface.monitoring.doneRewind )
   END_RUNG
   RUNG wire#powerrail
      Contact( #emFeedback.isLinked )
      Not()
      Coil( "Unit1.Em0.ControlNodes".unWinder.jobInterface.monitoring.doneLinkChg )
   END_RUNG
   // the same network as SCL:
   "Unit1.Em0.ControlNodes".unWinder.jobInterface.monitoring.doneRewind := NOT (NOT "Unit1.Em0.ControlNodes".unWinder."step".action[421]);
   "Unit1.Em0.ControlNodes".unWinder.jobInterface.monitoring.doneLinkChg := NOT #emFeedback.isLinked;
END_REGION

REGION Network 32: ******************** Control Modules (Axis) ********************
   // Call control modules that are actuators after the em logic (jobs and sequence), so that the latest commands are applied to the actuators.
END_REGION

REGION Network 33: Reset CMS
   RUNG wire#powerrail
      Contact( #statUnitStatus.acknowledgeActive )
      wire#w1
      Contact( "Unit1.Em0.ControlNodes".cmAirShaftOnOff.monitoring.error )
      Coil( "Unit1.Em0.ControlNodes".cmAirShaftOnOff.commands.reset )
   END_RUNG
   RUNG wire#powerrail
      Contact( #statUnitStatus.state.resetting )
   END_RUNG wire#w1
   RUNG wire#powerrail
      Contact( "Unit1.EmNodes".EnableACK )
   END_RUNG wire#w1
   RUNG wire#w1
      Contact( "Unit1.Em0.ControlNodes".cmExpelFwdBwd.monitoring.error )
      Coil( "Unit1.Em0.ControlNodes".cmExpelFwdBwd.commands.reset )
   END_RUNG
   RUNG wire#w1
      Contact( "Unit1.Em0.ControlNodes".cmRadiusMeasureAnalogInput.monitoring.error )
      Coil( "Unit1.Em0.ControlNodes".cmRadiusMeasureAnalogInput.commands.reset )
   END_RUNG
   RUNG wire#w1
      Contact( "Unit1.Em0.ControlNodes".cmEpc.monitoring.error )
      Coil( "Unit1.Em0.ControlNodes".cmEpc.commands.reset )
   END_RUNG
   RUNG wire#w1
      Contact( "Unit1.Em0.HmiInterface".cmBobinID.monitoring.error )
      Coil( "Unit1.Em0.HmiInterface".cmBobinID.commands.ResetReq )
   END_RUNG
   RUNG wire#powerrail
      Contact( #statUnitStatus.acknowledgeActive )
      wire#w2
      Contact( "Unit1.Em0.ControlNodes".cmUnWinderAxisB.monitoring.error )
      wire#w3
      Coil( "Unit1.Em0.ControlNodes".cmUnWinderAxisB.commands.resetAxis )
   END_RUNG
   RUNG wire#powerrail
      Contact( #statUnitStatus.state.resetting )
   END_RUNG wire#w2
   RUNG wire#powerrail
      Contact( "Unit1.EmNodes".EnableACK )
   END_RUNG wire#w2
   RUNG wire#w2
      Contact( "Unit1.Em0.ControlNodes".cmUnWinderAxisB.monitoring.statusWord1.Error )
   END_RUNG wire#w3
   RUNG wire#powerrail
      Contact( "Unit1.Em0.ControlNodes".cm.brakeTest.unwinder.commands.axisReset )
   END_RUNG wire#w3
   RUNG wire#w3
      I_Contact( "Unit1.Em0.ControlNodes".cmUnWinderAxisB.monitoring.axisEnabled )
      I_Contact( "Unit1.Em0.ControlNodes".cm.brakeTest.unwinder.commands.axisReset )
      Coil( "Unit1.Em0.ControlNodes".cmUnWinderAxisB.commandConfiguration.generalSettings.resetWithRestart )
   END_RUNG
   // the same network as SCL:
   #_w1 := #statUnitStatus.acknowledgeActive OR #statUnitStatus.state.resetting OR "Unit1.EmNodes".EnableACK;
   "Unit1.Em0.ControlNodes".cmAirShaftOnOff.commands.reset := #_w1 AND "Unit1.Em0.ControlNodes".cmAirShaftOnOff.monitoring.error;
   "Unit1.Em0.ControlNodes".cmExpelFwdBwd.commands.reset := #_w1 AND "Unit1.Em0.ControlNodes".cmExpelFwdBwd.monitoring.error;
   "Unit1.Em0.ControlNodes".cmRadiusMeasureAnalogInput.commands.reset := #_w1 AND "Unit1.Em0.ControlNodes".cmRadiusMeasureAnalogInput.monitoring.error;
   "Unit1.Em0.ControlNodes".cmEpc.commands.reset := #_w1 AND "Unit1.Em0.ControlNodes".cmEpc.monitoring.error;
   "Unit1.Em0.HmiInterface".cmBobinID.commands.ResetReq := #_w1 AND "Unit1.Em0.HmiInterface".cmBobinID.monitoring.error;
   "Unit1.Em0.ControlNodes".cmUnWinderAxisB.commands.resetAxis := ((#statUnitStatus.acknowledgeActive OR #statUnitStatus.state.resetting OR "Unit1.EmNodes".EnableACK) AND ("Unit1.Em0.ControlNodes".cmUnWinderAxisB.monitoring.error OR "Unit1.Em0.ControlNodes".cmUnWinderAxisB.monitoring.statusWord1.Error)) OR "Unit1.Em0.ControlNodes".cm.brakeTest.unwinder.commands.axisReset;
   "Unit1.Em0.ControlNodes".cmUnWinderAxisB.commandConfiguration.generalSettings.resetWithRestart := "Unit1.Em0.ControlNodes".cmUnWinderAxisB.commands.resetAxis AND NOT "Unit1.Em0.ControlNodes".cmUnWinderAxisB.monitoring.axisEnabled AND NOT "Unit1.Em0.ControlNodes".cm.brakeTest.unwinder.commands.axisReset;
END_REGION

REGION Network 34: Enable/Disable CMs
   // Enable the axis during the resetting state and disable the axis during the aborting state.
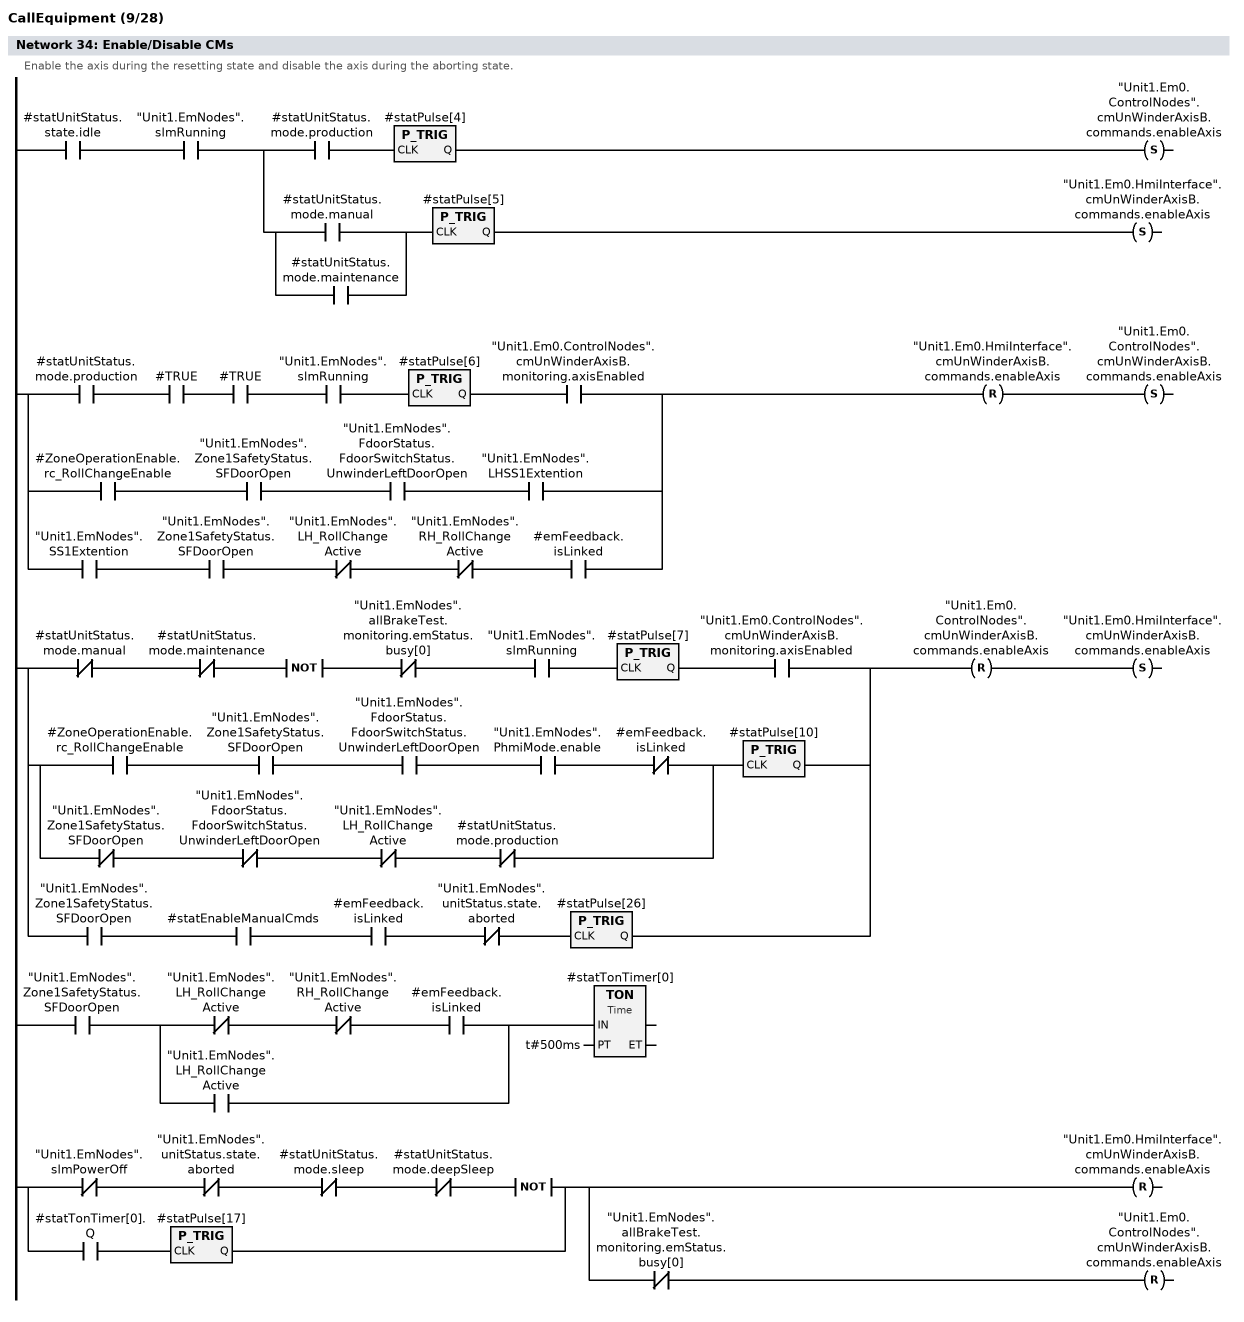
   RUNG wire#powerrail
      Contact( #statUnitStatus.state.idle )
      Contact( "Unit1.EmNodes".slmRunning )
      wire#w1
      Contact( #statUnitStatus.mode.production )
      P_Trig( #statPulse[4] )
      S_Coil( "Unit1.Em0.ControlNodes".cmUnWinderAxisB.commands.enableAxis )
   END_RUNG
   RUNG wire#w1
      Contact( #statUnitStatus.mode.manual )
      wire#w2
      P_Trig( #statPulse[5] )
      S_Coil( "Unit1.Em0.HmiInterface".cmUnWinderAxisB.commands.enableAxis )
   END_RUNG
   RUNG wire#w1
      Contact( #statUnitStatus.mode.maintenance )
   END_RUNG wire#w2
   RUNG wire#powerrail
      Contact( #statUnitStatus.mode.production )
      Contact( #TRUE )
      Contact( #TRUE )
      Contact( "Unit1.EmNodes".slmRunning )
      P_Trig( #statPulse[6] )
      Contact( "Unit1.Em0.ControlNodes".cmUnWinderAxisB.monitoring.axisEnabled )
      wire#w3
      R_Coil( "Unit1.Em0.HmiInterface".cmUnWinderAxisB.commands.enableAxis )
      S_Coil( "Unit1.Em0.ControlNodes".cmUnWinderAxisB.commands.enableAxis )
   END_RUNG
   RUNG wire#powerrail
      Contact( #ZoneOperationEnable.rc_RollChangeEnable )
      Contact( "Unit1.EmNodes".Zone1SafetyStatus.SFDoorOpen )
      Contact( "Unit1.EmNodes".FdoorStatus.FdoorSwitchStatus.UnwinderLeftDoorOpen )
      Contact( "Unit1.EmNodes".LHSS1Extention )
   END_RUNG wire#w3
   RUNG wire#powerrail
      Contact( "Unit1.EmNodes".SS1Extention )
      Contact( "Unit1.EmNodes".Zone1SafetyStatus.SFDoorOpen )
      I_Contact( "Unit1.EmNodes".LH_RollChangeActive )
      I_Contact( "Unit1.EmNodes".RH_RollChangeActive )
      Contact( #emFeedback.isLinked )
   END_RUNG wire#w3
   RUNG wire#powerrail
      I_Contact( #statUnitStatus.mode.manual )
      I_Contact( #statUnitStatus.mode.maintenance )
      Not()
      I_Contact( "Unit1.EmNodes".allBrakeTest.monitoring.emStatus.busy[0] )
      Contact( "Unit1.EmNodes".slmRunning )
      P_Trig( #statPulse[7] )
      Contact( "Unit1.Em0.ControlNodes".cmUnWinderAxisB.monitoring.axisEnabled )
      wire#w4
      R_Coil( "Unit1.Em0.ControlNodes".cmUnWinderAxisB.commands.enableAxis )
      S_Coil( "Unit1.Em0.HmiInterface".cmUnWinderAxisB.commands.enableAxis )
   END_RUNG
   RUNG wire#powerrail
      Contact( #ZoneOperationEnable.rc_RollChangeEnable )
      Contact( "Unit1.EmNodes".Zone1SafetyStatus.SFDoorOpen )
      Contact( "Unit1.EmNodes".FdoorStatus.FdoorSwitchStatus.UnwinderLeftDoorOpen )
      Contact( "Unit1.EmNodes".PhmiMode.enable )
      I_Contact( #emFeedback.isLinked )
      wire#w5
      P_Trig( #statPulse[10] )
   END_RUNG wire#w4
   RUNG wire#powerrail
      I_Contact( "Unit1.EmNodes".Zone1SafetyStatus.SFDoorOpen )
      I_Contact( "Unit1.EmNodes".FdoorStatus.FdoorSwitchStatus.UnwinderLeftDoorOpen )
      I_Contact( "Unit1.EmNodes".LH_RollChangeActive )
      I_Contact( #statUnitStatus.mode.production )
   END_RUNG wire#w5
   RUNG wire#powerrail
      Contact( "Unit1.EmNodes".Zone1SafetyStatus.SFDoorOpen )
      Contact( #statEnableManualCmds )
      Contact( #emFeedback.isLinked )
      I_Contact( "Unit1.EmNodes".unitStatus.state.aborted )
      P_Trig( #statPulse[26] )
   END_RUNG wire#w4
   RUNG wire#powerrail
      Contact( "Unit1.EmNodes".Zone1SafetyStatus.SFDoorOpen )
      wire#w6
      I_Contact( "Unit1.EmNodes".LH_RollChangeActive )
      I_Contact( "Unit1.EmNodes".RH_RollChangeActive )
      Contact( #emFeedback.isLinked )
      wire#w7
      { S7_Templates := "time_type := Time" } #statTonTimer[0].TON(pt := t#500ms, et =>)
   END_RUNG
   RUNG wire#w6
      Contact( "Unit1.EmNodes".LH_RollChangeActive )
   END_RUNG wire#w7
   RUNG wire#powerrail
      I_Contact( "Unit1.EmNodes".slmPowerOff )
      I_Contact( "Unit1.EmNodes".unitStatus.state.aborted )
      I_Contact( #statUnitStatus.mode.sleep )
      I_Contact( #statUnitStatus.mode.deepSleep )
      Not()
      wire#w8
      R_Coil( "Unit1.Em0.HmiInterface".cmUnWinderAxisB.commands.enableAxis )
   END_RUNG
   RUNG wire#powerrail
      Contact( #statTonTimer[0].Q )
      P_Trig( #statPulse[17] )
   END_RUNG wire#w8
   RUNG wire#w8
      I_Contact( "Unit1.EmNodes".allBrakeTest.monitoring.emStatus.busy[0] )
      R_Coil( "Unit1.Em0.ControlNodes".cmUnWinderAxisB.commands.enableAxis )
   END_RUNG
   // the same network as SCL:
   #_w1 := #statUnitStatus.state.idle AND "Unit1.EmNodes".slmRunning;
   #_w2 := #_w1 AND #statUnitStatus.mode.production;
   #_w3 := #_w2 AND NOT #statPulse[4];   // rising edge
   #statPulse[4] := #_w2;
   IF #_w3 THEN "Unit1.Em0.ControlNodes".cmUnWinderAxisB.commands.enableAxis := TRUE; END_IF;
   #_w4 := #_w1 AND (#statUnitStatus.mode.manual OR #statUnitStatus.mode.maintenance);
   #_w5 := #_w4 AND NOT #statPulse[5];   // rising edge
   #statPulse[5] := #_w4;
   IF #_w5 THEN "Unit1.Em0.HmiInterface".cmUnWinderAxisB.commands.enableAxis := TRUE; END_IF;
   #_w6 := #statUnitStatus.mode.production AND #TRUE AND #TRUE AND "Unit1.EmNodes".slmRunning;
   #_w7 := #_w6 AND NOT #statPulse[6];   // rising edge
   #statPulse[6] := #_w6;
   IF (#_w7 AND "Unit1.Em0.ControlNodes".cmUnWinderAxisB.monitoring.axisEnabled) OR (#ZoneOperationEnable.rc_RollChangeEnable AND "Unit1.EmNodes".Zone1SafetyStatus.SFDoorOpen AND "Unit1.EmNodes".FdoorStatus.FdoorSwitchStatus.UnwinderLeftDoorOpen AND "Unit1.EmNodes".LHSS1Extention) OR ("Unit1.EmNodes".SS1Extention AND "Unit1.EmNodes".Zone1SafetyStatus.SFDoorOpen AND NOT "Unit1.EmNodes".LH_RollChangeActive AND NOT "Unit1.EmNodes".RH_RollChangeActive AND #emFeedback.isLinked) THEN
       "Unit1.Em0.HmiInterface".cmUnWinderAxisB.commands.enableAxis := FALSE;
       "Unit1.Em0.ControlNodes".cmUnWinderAxisB.commands.enableAxis := TRUE;
   END_IF;
   #_w8 := NOT (NOT #statUnitStatus.mode.manual AND NOT #statUnitStatus.mode.maintenance) AND NOT "Unit1.EmNodes".allBrakeTest.monitoring.emStatus.busy[0] AND "Unit1.EmNodes".slmRunning;
   #_w9 := #_w8 AND NOT #statPulse[7];   // rising edge
   #statPulse[7] := #_w8;
   #_w10 := (#ZoneOperationEnable.rc_RollChangeEnable AND "Unit1.EmNodes".Zone1SafetyStatus.SFDoorOpen AND "Unit1.EmNodes".FdoorStatus.FdoorSwitchStatus.UnwinderLeftDoorOpen AND "Unit1.EmNodes".PhmiMode.enable AND NOT #emFeedback.isLinked) OR (NOT "Unit1.EmNodes".Zone1SafetyStatus.SFDoorOpen AND NOT "Unit1.EmNodes".FdoorStatus.FdoorSwitchStatus.UnwinderLeftDoorOpen AND NOT "Unit1.EmNodes".LH_RollChangeActive AND NOT #statUnitStatus.mode.production);
   #_w11 := #_w10 AND NOT #statPulse[10];   // rising edge
   #statPulse[10] := #_w10;
   #_w12 := "Unit1.EmNodes".Zone1SafetyStatus.SFDoorOpen AND #statEnableManualCmds AND #emFeedback.isLinked AND NOT "Unit1.EmNodes".unitStatus.state.aborted;
   #_w13 := #_w12 AND NOT #statPulse[26];   // rising edge
   #statPulse[26] := #_w12;
   IF (#_w9 AND "Unit1.Em0.ControlNodes".cmUnWinderAxisB.monitoring.axisEnabled) OR #_w11 OR #_w13 THEN
       "Unit1.Em0.ControlNodes".cmUnWinderAxisB.commands.enableAxis := FALSE;
       "Unit1.Em0.HmiInterface".cmUnWinderAxisB.commands.enableAxis := TRUE;
   END_IF;
   #statTonTimer[0].TON(IN := "Unit1.EmNodes".Zone1SafetyStatus.SFDoorOpen AND ((NOT "Unit1.EmNodes".LH_RollChangeActive AND NOT "Unit1.EmNodes".RH_RollChangeActive AND #emFeedback.isLinked) OR "Unit1.EmNodes".LH_RollChangeActive),
                        PT := t#500ms);
   #_w14 := #statTonTimer[0].Q AND NOT #statPulse[17];   // rising edge
   #statPulse[17] := #statTonTimer[0].Q;
   #_w15 := NOT (NOT "Unit1.EmNodes".slmPowerOff AND NOT "Unit1.EmNodes".unitStatus.state.aborted AND NOT #statUnitStatus.mode.sleep AND NOT #statUnitStatus.mode.deepSleep) OR #_w14;
   IF #_w15 THEN "Unit1.Em0.HmiInterface".cmUnWinderAxisB.commands.enableAxis := FALSE; END_IF;
   IF #_w15 AND NOT "Unit1.EmNodes".allBrakeTest.monitoring.emStatus.busy[0] THEN
       "Unit1.Em0.ControlNodes".cmUnWinderAxisB.commands.enableAxis := FALSE;
   END_IF;
END_REGION

REGION Network 35: CM UnWinder B Axis Command Jog
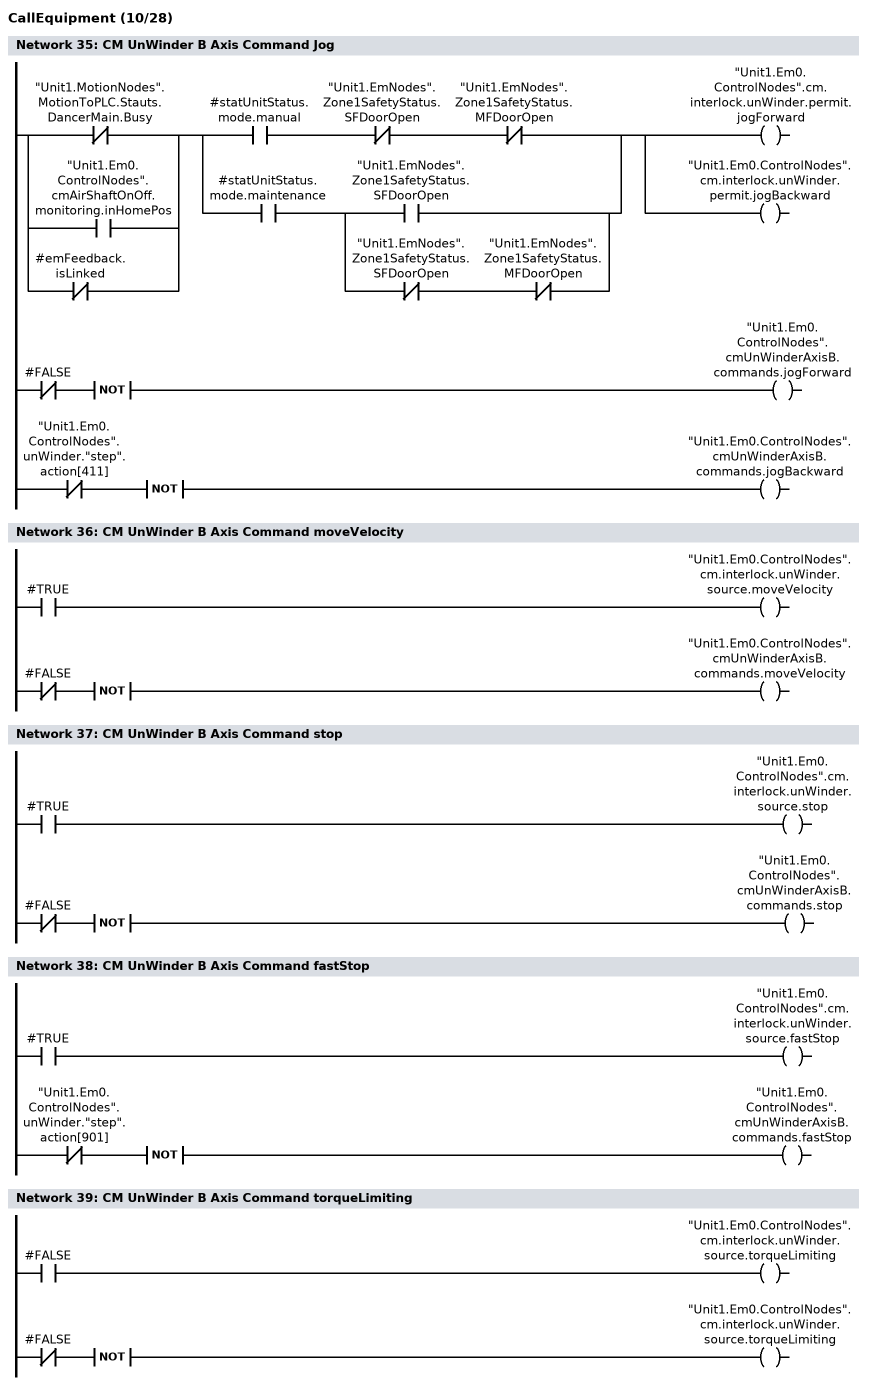
   RUNG wire#powerrail
      I_Contact( "Unit1.MotionNodes".MotionToPLC.Stauts.DancerMain.Busy )
      wire#w1
      Contact( #statUnitStatus.mode.manual )
      I_Contact( "Unit1.EmNodes".Zone1SafetyStatus.SFDoorOpen )
      I_Contact( "Unit1.EmNodes".Zone1SafetyStatus.MFDoorOpen )
      wire#w2
      Coil( "Unit1.Em0.ControlNodes".cm.interlock.unWinder.permit.jogForward )
   END_RUNG
   RUNG wire#powerrail
      Contact( "Unit1.Em0.ControlNodes".cmAirShaftOnOff.monitoring.inHomePos )
   END_RUNG wire#w1
   RUNG wire#powerrail
      I_Contact( #emFeedback.isLinked )
   END_RUNG wire#w1
   RUNG wire#w1
      Contact( #statUnitStatus.mode.maintenance )
      wire#w3
      Contact( "Unit1.EmNodes".Zone1SafetyStatus.SFDoorOpen )
   END_RUNG wire#w2
   RUNG wire#w3
      I_Contact( "Unit1.EmNodes".Zone1SafetyStatus.SFDoorOpen )
      I_Contact( "Unit1.EmNodes".Zone1SafetyStatus.MFDoorOpen )
   END_RUNG wire#w2
   RUNG wire#w2
      Coil( "Unit1.Em0.ControlNodes".cm.interlock.unWinder.permit.jogBackward )
   END_RUNG
   RUNG wire#powerrail
      I_Contact( #FALSE )
      Not()
      Coil( "Unit1.Em0.ControlNodes".cmUnWinderAxisB.commands.jogForward )
   END_RUNG
   RUNG wire#powerrail
      I_Contact( "Unit1.Em0.ControlNodes".unWinder."step".action[411] )
      Not()
      Coil( "Unit1.Em0.ControlNodes".cmUnWinderAxisB.commands.jogBackward )
   END_RUNG
   // the same network as SCL:
   "Unit1.Em0.ControlNodes".cm.interlock.unWinder.permit.jogForward := (NOT "Unit1.MotionNodes".MotionToPLC.Stauts.DancerMain.Busy OR "Unit1.Em0.ControlNodes".cmAirShaftOnOff.monitoring.inHomePos OR NOT #emFeedback.isLinked) AND ((#statUnitStatus.mode.manual AND NOT "Unit1.EmNodes".Zone1SafetyStatus.SFDoorOpen AND NOT "Unit1.EmNodes".Zone1SafetyStatus.MFDoorOpen) OR (#statUnitStatus.mode.maintenance AND ("Unit1.EmNodes".Zone1SafetyStatus.SFDoorOpen OR (NOT "Unit1.EmNodes".Zone1SafetyStatus.SFDoorOpen AND NOT "Unit1.EmNodes".Zone1SafetyStatus.MFDoorOpen))));
   "Unit1.Em0.ControlNodes".cm.interlock.unWinder.permit.jogBackward := "Unit1.Em0.ControlNodes".cm.interlock.unWinder.permit.jogForward;
   "Unit1.Em0.ControlNodes".cmUnWinderAxisB.commands.jogForward := NOT (NOT #FALSE);
   "Unit1.Em0.ControlNodes".cmUnWinderAxisB.commands.jogBackward := NOT (NOT "Unit1.Em0.ControlNodes".unWinder."step".action[411]);
END_REGION

REGION Network 36: CM UnWinder B Axis Command moveVelocity
   RUNG wire#powerrail
      Contact( #TRUE )
      Coil( "Unit1.Em0.ControlNodes".cm.interlock.unWinder.source.moveVelocity )
   END_RUNG
   RUNG wire#powerrail
      I_Contact( #FALSE )
      Not()
      Coil( "Unit1.Em0.ControlNodes".cmUnWinderAxisB.commands.moveVelocity )
   END_RUNG
   // the same network as SCL:
   "Unit1.Em0.ControlNodes".cm.interlock.unWinder.source.moveVelocity := #TRUE;
   "Unit1.Em0.ControlNodes".cmUnWinderAxisB.commands.moveVelocity := NOT (NOT #FALSE);
END_REGION

REGION Network 37: CM UnWinder B Axis Command stop
   RUNG wire#powerrail
      Contact( #TRUE )
      Coil( "Unit1.Em0.ControlNodes".cm.interlock.unWinder.source.stop )
   END_RUNG
   RUNG wire#powerrail
      I_Contact( #FALSE )
      Not()
      Coil( "Unit1.Em0.ControlNodes".cmUnWinderAxisB.commands.stop )
   END_RUNG
   // the same network as SCL:
   "Unit1.Em0.ControlNodes".cm.interlock.unWinder.source.stop := #TRUE;
   "Unit1.Em0.ControlNodes".cmUnWinderAxisB.commands.stop := NOT (NOT #FALSE);
END_REGION

REGION Network 38: CM UnWinder B Axis Command fastStop
   RUNG wire#powerrail
      Contact( #TRUE )
      Coil( "Unit1.Em0.ControlNodes".cm.interlock.unWinder.source.fastStop )
   END_RUNG
   RUNG wire#powerrail
      I_Contact( "Unit1.Em0.ControlNodes".unWinder."step".action[901] )
      Not()
      Coil( "Unit1.Em0.ControlNodes".cmUnWinderAxisB.commands.fastStop )
   END_RUNG
   // the same network as SCL:
   "Unit1.Em0.ControlNodes".cm.interlock.unWinder.source.fastStop := #TRUE;
   "Unit1.Em0.ControlNodes".cmUnWinderAxisB.commands.fastStop := NOT (NOT "Unit1.Em0.ControlNodes".unWinder."step".action[901]);
END_REGION

REGION Network 39: CM UnWinder B Axis Command torqueLimiting
   RUNG wire#powerrail
      Contact( #FALSE )
      Coil( "Unit1.Em0.ControlNodes".cm.interlock.unWinder.source.torqueLimiting )
   END_RUNG
   RUNG wire#powerrail
      I_Contact( #FALSE )
      Not()
      Coil( "Unit1.Em0.ControlNodes".cm.interlock.unWinder.source.torqueLimiting )
   END_RUNG
   // the same network as SCL:
   "Unit1.Em0.ControlNodes".cm.interlock.unWinder.source.torqueLimiting := #FALSE;
   "Unit1.Em0.ControlNodes".cm.interlock.unWinder.source.torqueLimiting := NOT (NOT #FALSE);
END_REGION

REGION Network 40: CM UnWinder B Axis Command homing
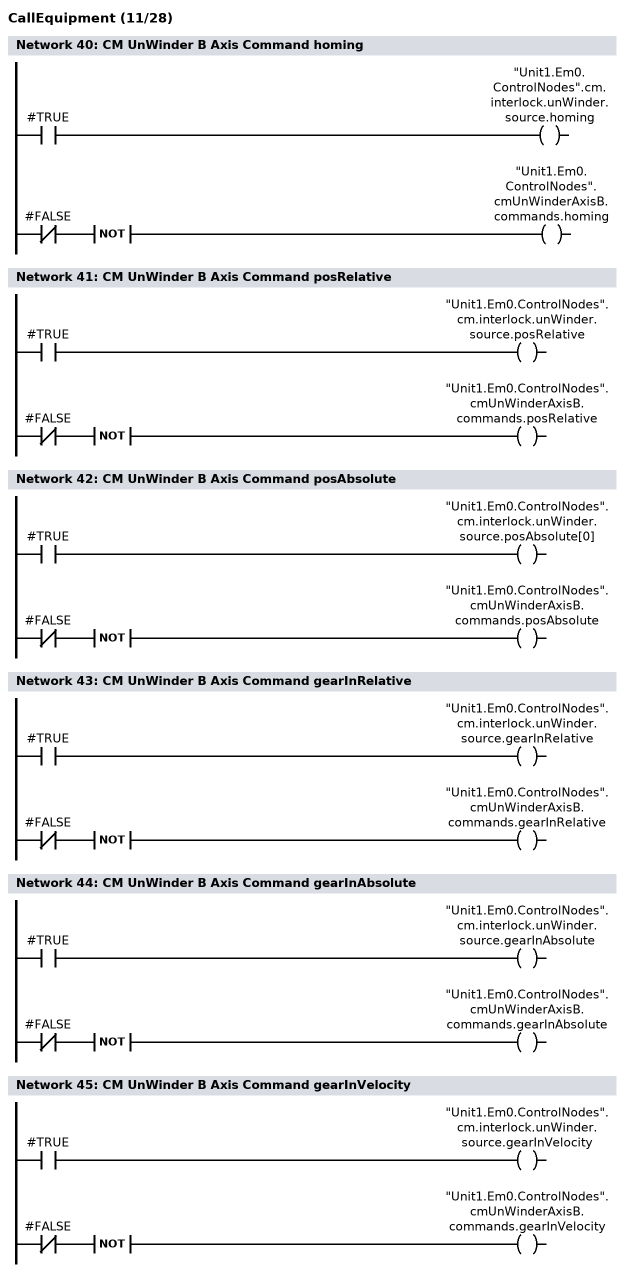
   RUNG wire#powerrail
      Contact( #TRUE )
      Coil( "Unit1.Em0.ControlNodes".cm.interlock.unWinder.source.homing )
   END_RUNG
   RUNG wire#powerrail
      I_Contact( #FALSE )
      Not()
      Coil( "Unit1.Em0.ControlNodes".cmUnWinderAxisB.commands.homing )
   END_RUNG
   // the same network as SCL:
   "Unit1.Em0.ControlNodes".cm.interlock.unWinder.source.homing := #TRUE;
   "Unit1.Em0.ControlNodes".cmUnWinderAxisB.commands.homing := NOT (NOT #FALSE);
END_REGION

REGION Network 41: CM UnWinder B Axis Command posRelative
   RUNG wire#powerrail
      Contact( #TRUE )
      Coil( "Unit1.Em0.ControlNodes".cm.interlock.unWinder.source.posRelative )
   END_RUNG
   RUNG wire#powerrail
      I_Contact( #FALSE )
      Not()
      Coil( "Unit1.Em0.ControlNodes".cmUnWinderAxisB.commands.posRelative )
   END_RUNG
   // the same network as SCL:
   "Unit1.Em0.ControlNodes".cm.interlock.unWinder.source.posRelative := #TRUE;
   "Unit1.Em0.ControlNodes".cmUnWinderAxisB.commands.posRelative := NOT (NOT #FALSE);
END_REGION

REGION Network 42: CM UnWinder B Axis Command posAbsolute
   RUNG wire#powerrail
      Contact( #TRUE )
      Coil( "Unit1.Em0.ControlNodes".cm.interlock.unWinder.source.posAbsolute[0] )
   END_RUNG
   RUNG wire#powerrail
      I_Contact( #FALSE )
      Not()
      Coil( "Unit1.Em0.ControlNodes".cmUnWinderAxisB.commands.posAbsolute )
   END_RUNG
   // the same network as SCL:
   "Unit1.Em0.ControlNodes".cm.interlock.unWinder.source.posAbsolute[0] := #TRUE;
   "Unit1.Em0.ControlNodes".cmUnWinderAxisB.commands.posAbsolute := NOT (NOT #FALSE);
END_REGION

REGION Network 43: CM UnWinder B Axis Command gearInRelative
   RUNG wire#powerrail
      Contact( #TRUE )
      Coil( "Unit1.Em0.ControlNodes".cm.interlock.unWinder.source.gearInRelative )
   END_RUNG
   RUNG wire#powerrail
      I_Contact( #FALSE )
      Not()
      Coil( "Unit1.Em0.ControlNodes".cmUnWinderAxisB.commands.gearInRelative )
   END_RUNG
   // the same network as SCL:
   "Unit1.Em0.ControlNodes".cm.interlock.unWinder.source.gearInRelative := #TRUE;
   "Unit1.Em0.ControlNodes".cmUnWinderAxisB.commands.gearInRelative := NOT (NOT #FALSE);
END_REGION

REGION Network 44: CM UnWinder B Axis Command gearInAbsolute
   RUNG wire#powerrail
      Contact( #TRUE )
      Coil( "Unit1.Em0.ControlNodes".cm.interlock.unWinder.source.gearInAbsolute )
   END_RUNG
   RUNG wire#powerrail
      I_Contact( #FALSE )
      Not()
      Coil( "Unit1.Em0.ControlNodes".cmUnWinderAxisB.commands.gearInAbsolute )
   END_RUNG
   // the same network as SCL:
   "Unit1.Em0.ControlNodes".cm.interlock.unWinder.source.gearInAbsolute := #TRUE;
   "Unit1.Em0.ControlNodes".cmUnWinderAxisB.commands.gearInAbsolute := NOT (NOT #FALSE);
END_REGION

REGION Network 45: CM UnWinder B Axis Command gearInVelocity
   RUNG wire#powerrail
      Contact( #TRUE )
      Coil( "Unit1.Em0.ControlNodes".cm.interlock.unWinder.source.gearInVelocity )
   END_RUNG
   RUNG wire#powerrail
      I_Contact( #FALSE )
      Not()
      Coil( "Unit1.Em0.ControlNodes".cmUnWinderAxisB.commands.gearInVelocity )
   END_RUNG
   // the same network as SCL:
   "Unit1.Em0.ControlNodes".cm.interlock.unWinder.source.gearInVelocity := #TRUE;
   "Unit1.Em0.ControlNodes".cmUnWinderAxisB.commands.gearInVelocity := NOT (NOT #FALSE);
END_REGION

REGION Network 46: CM UnWinder B Axis Command camIn
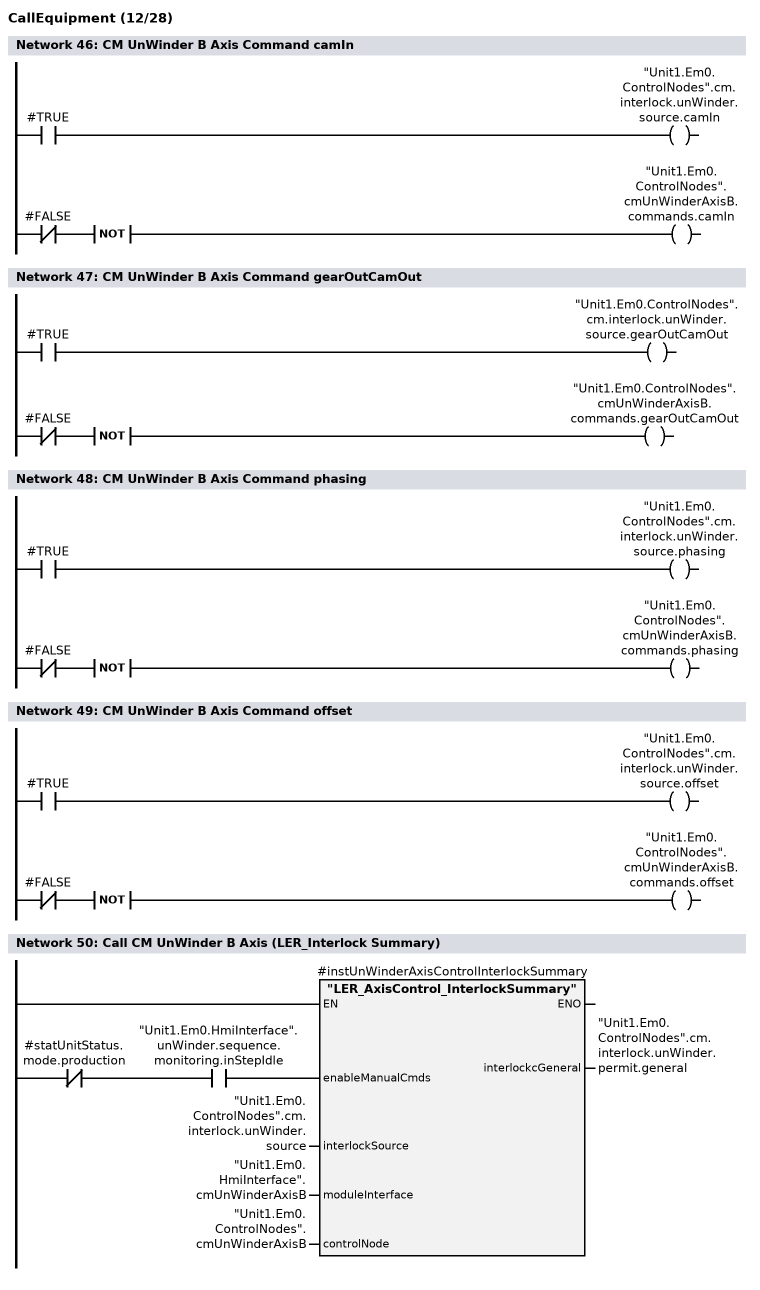
   RUNG wire#powerrail
      Contact( #TRUE )
      Coil( "Unit1.Em0.ControlNodes".cm.interlock.unWinder.source.camIn )
   END_RUNG
   RUNG wire#powerrail
      I_Contact( #FALSE )
      Not()
      Coil( "Unit1.Em0.ControlNodes".cmUnWinderAxisB.commands.camIn )
   END_RUNG
   // the same network as SCL:
   "Unit1.Em0.ControlNodes".cm.interlock.unWinder.source.camIn := #TRUE;
   "Unit1.Em0.ControlNodes".cmUnWinderAxisB.commands.camIn := NOT (NOT #FALSE);
END_REGION

REGION Network 47: CM UnWinder B Axis Command gearOutCamOut
   RUNG wire#powerrail
      Contact( #TRUE )
      Coil( "Unit1.Em0.ControlNodes".cm.interlock.unWinder.source.gearOutCamOut )
   END_RUNG
   RUNG wire#powerrail
      I_Contact( #FALSE )
      Not()
      Coil( "Unit1.Em0.ControlNodes".cmUnWinderAxisB.commands.gearOutCamOut )
   END_RUNG
   // the same network as SCL:
   "Unit1.Em0.ControlNodes".cm.interlock.unWinder.source.gearOutCamOut := #TRUE;
   "Unit1.Em0.ControlNodes".cmUnWinderAxisB.commands.gearOutCamOut := NOT (NOT #FALSE);
END_REGION

REGION Network 48: CM UnWinder B Axis Command phasing
   RUNG wire#powerrail
      Contact( #TRUE )
      Coil( "Unit1.Em0.ControlNodes".cm.interlock.unWinder.source.phasing )
   END_RUNG
   RUNG wire#powerrail
      I_Contact( #FALSE )
      Not()
      Coil( "Unit1.Em0.ControlNodes".cmUnWinderAxisB.commands.phasing )
   END_RUNG
   // the same network as SCL:
   "Unit1.Em0.ControlNodes".cm.interlock.unWinder.source.phasing := #TRUE;
   "Unit1.Em0.ControlNodes".cmUnWinderAxisB.commands.phasing := NOT (NOT #FALSE);
END_REGION

REGION Network 49: CM UnWinder B Axis Command offset
   RUNG wire#powerrail
      Contact( #TRUE )
      Coil( "Unit1.Em0.ControlNodes".cm.interlock.unWinder.source.offset )
   END_RUNG
   RUNG wire#powerrail
      I_Contact( #FALSE )
      Not()
      Coil( "Unit1.Em0.ControlNodes".cmUnWinderAxisB.commands.offset )
   END_RUNG
   // the same network as SCL:
   "Unit1.Em0.ControlNodes".cm.interlock.unWinder.source.offset := #TRUE;
   "Unit1.Em0.ControlNodes".cmUnWinderAxisB.commands.offset := NOT (NOT #FALSE);
END_REGION

REGION Network 50: Call CM UnWinder B Axis (LER_Interlock Summary)
   RUNG wire#powerrail
      #instUnWinderAxisControlInterlockSummary(enableManualCmds := wire#w1, interlockSource := "Unit1.Em0.ControlNodes".cm.interlock.unWinder.source, moduleInterface := "Unit1.Em0.HmiInterface".cmUnWinderAxisB, controlNode := "Unit1.Em0.ControlNodes".cmUnWinderAxisB, interlockcGeneral => "Unit1.Em0.ControlNodes".cm.interlock.unWinder.permit.general)
   END_RUNG
   RUNG wire#powerrail
      I_Contact( #statUnitStatus.mode.production )
      Contact( "Unit1.Em0.HmiInterface".unWinder.sequence.monitoring.inStepIdle )
   END_RUNG wire#w1
   // the same network as SCL:
   #instUnWinderAxisControlInterlockSummary(enableManualCmds := NOT #statUnitStatus.mode.production AND "Unit1.Em0.HmiInterface".unWinder.sequence.monitoring.inStepIdle,   // "LER_AxisControl_InterlockSummary"
                           interlockSource := "Unit1.Em0.ControlNodes".cm.interlock.unWinder.source,
                           moduleInterface := "Unit1.Em0.HmiInterface".cmUnWinderAxisB,
                           controlNode := "Unit1.Em0.ControlNodes".cmUnWinderAxisB,
                           interlockcGeneral => "Unit1.Em0.ControlNodes".cm.interlock.unWinder.permit.general);
END_REGION

REGION Network 51: SpeedLimitByRadius
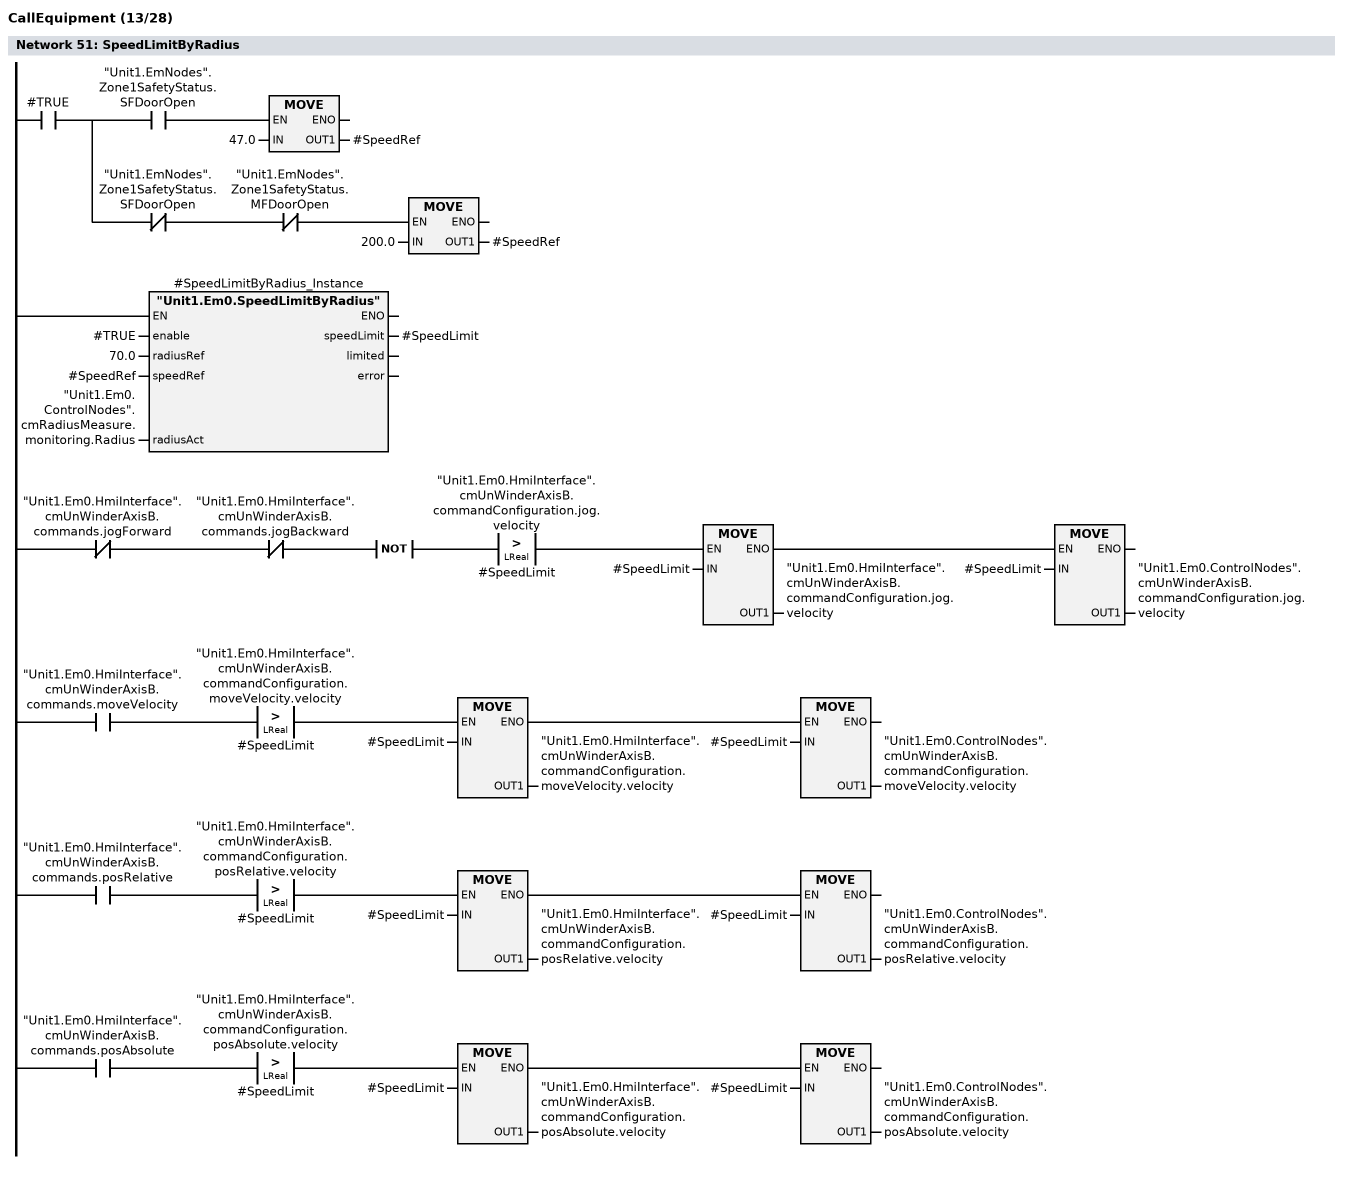
   RUNG wire#powerrail
      Contact( #TRUE )
      wire#w1
      Contact( "Unit1.EmNodes".Zone1SafetyStatus.SFDoorOpen )
      Move(in := 47.0, out1 => #SpeedRef)
   END_RUNG
   RUNG wire#w1
      I_Contact( "Unit1.EmNodes".Zone1SafetyStatus.SFDoorOpen )
      I_Contact( "Unit1.EmNodes".Zone1SafetyStatus.MFDoorOpen )
      Move(in := 200.0, out1 => #SpeedRef)
   END_RUNG
   RUNG wire#powerrail
      #SpeedLimitByRadius_Instance(enable := #TRUE, radiusRef := 70.0, speedRef := #SpeedRef, radiusAct := "Unit1.Em0.ControlNodes".cmRadiusMeasure.monitoring.Radius, speedLimit => #SpeedLimit, limited =>, error =>)
   END_RUNG
   RUNG wire#powerrail
      I_Contact( "Unit1.Em0.HmiInterface".cmUnWinderAxisB.commands.jogForward )
      I_Contact( "Unit1.Em0.HmiInterface".cmUnWinderAxisB.commands.jogBackward )
      Not()
      { S7_Templates := "SrcType := LReal" } GT_Contact(in1 := "Unit1.Em0.HmiInterface".cmUnWinderAxisB.commandConfiguration.jog.velocity, in2 := #SpeedLimit)
      Move(in := #SpeedLimit, out1 => "Unit1.Em0.HmiInterface".cmUnWinderAxisB.commandConfiguration.jog.velocity)
      Move(in := #SpeedLimit, out1 => "Unit1.Em0.ControlNodes".cmUnWinderAxisB.commandConfiguration.jog.velocity)
   END_RUNG
   RUNG wire#powerrail
      Contact( "Unit1.Em0.HmiInterface".cmUnWinderAxisB.commands.moveVelocity )
      { S7_Templates := "SrcType := LReal" } GT_Contact(in1 := "Unit1.Em0.HmiInterface".cmUnWinderAxisB.commandConfiguration.moveVelocity.velocity, in2 := #SpeedLimit)
      Move(in := #SpeedLimit, out1 => "Unit1.Em0.HmiInterface".cmUnWinderAxisB.commandConfiguration.moveVelocity.velocity)
      Move(in := #SpeedLimit, out1 => "Unit1.Em0.ControlNodes".cmUnWinderAxisB.commandConfiguration.moveVelocity.velocity)
   END_RUNG
   RUNG wire#powerrail
      Contact( "Unit1.Em0.HmiInterface".cmUnWinderAxisB.commands.posRelative )
      { S7_Templates := "SrcType := LReal" } GT_Contact(in1 := "Unit1.Em0.HmiInterface".cmUnWinderAxisB.commandConfiguration.posRelative.velocity, in2 := #SpeedLimit)
      Move(in := #SpeedLimit, out1 => "Unit1.Em0.HmiInterface".cmUnWinderAxisB.commandConfiguration.posRelative.velocity)
      Move(in := #SpeedLimit, out1 => "Unit1.Em0.ControlNodes".cmUnWinderAxisB.commandConfiguration.posRelative.velocity)
   END_RUNG
   RUNG wire#powerrail
      Contact( "Unit1.Em0.HmiInterface".cmUnWinderAxisB.commands.posAbsolute )
      { S7_Templates := "SrcType := LReal" } GT_Contact(in1 := "Unit1.Em0.HmiInterface".cmUnWinderAxisB.commandConfiguration.posAbsolute.velocity, in2 := #SpeedLimit)
      Move(in := #SpeedLimit, out1 => "Unit1.Em0.HmiInterface".cmUnWinderAxisB.commandConfiguration.posAbsolute.velocity)
      Move(in := #SpeedLimit, out1 => "Unit1.Em0.ControlNodes".cmUnWinderAxisB.commandConfiguration.posAbsolute.velocity)
   END_RUNG
   // the same network as SCL:
   IF #TRUE AND "Unit1.EmNodes".Zone1SafetyStatus.SFDoorOpen THEN #SpeedRef := 47.0; END_IF;
   IF #TRUE AND NOT "Unit1.EmNodes".Zone1SafetyStatus.SFDoorOpen AND NOT "Unit1.EmNodes".Zone1SafetyStatus.MFDoorOpen THEN
       #SpeedRef := 200.0;
   END_IF;
   #SpeedLimitByRadius_Instance(enable := #TRUE,   // "Unit1.Em0.SpeedLimitByRadius"
                           radiusRef := 70.0,
                           speedRef := #SpeedRef,
                           radiusAct := "Unit1.Em0.ControlNodes".cmRadiusMeasure.monitoring.Radius,
                           speedLimit => #SpeedLimit);
   #_w1 := NOT (NOT "Unit1.Em0.HmiInterface".cmUnWinderAxisB.commands.jogForward AND NOT "Unit1.Em0.HmiInterface".cmUnWinderAxisB.commands.jogBackward) AND ("Unit1.Em0.HmiInterface".cmUnWinderAxisB.commandConfiguration.jog.velocity > #SpeedLimit);
   IF #_w1 THEN
       "Unit1.Em0.HmiInterface".cmUnWinderAxisB.commandConfiguration.jog.velocity := #SpeedLimit;
       "Unit1.Em0.ControlNodes".cmUnWinderAxisB.commandConfiguration.jog.velocity := #SpeedLimit;
   END_IF;
   #_w2 := "Unit1.Em0.HmiInterface".cmUnWinderAxisB.commands.moveVelocity AND ("Unit1.Em0.HmiInterface".cmUnWinderAxisB.commandConfiguration.moveVelocity.velocity > #SpeedLimit);
   IF #_w2 THEN
       "Unit1.Em0.HmiInterface".cmUnWinderAxisB.commandConfiguration.moveVelocity.velocity := #SpeedLimit;
       "Unit1.Em0.ControlNodes".cmUnWinderAxisB.commandConfiguration.moveVelocity.velocity := #SpeedLimit;
   END_IF;
   #_w3 := "Unit1.Em0.HmiInterface".cmUnWinderAxisB.commands.posRelative AND ("Unit1.Em0.HmiInterface".cmUnWinderAxisB.commandConfiguration.posRelative.velocity > #SpeedLimit);
   IF #_w3 THEN
       "Unit1.Em0.HmiInterface".cmUnWinderAxisB.commandConfiguration.posRelative.velocity := #SpeedLimit;
       "Unit1.Em0.ControlNodes".cmUnWinderAxisB.commandConfiguration.posRelative.velocity := #SpeedLimit;
   END_IF;
   #_w4 := "Unit1.Em0.HmiInterface".cmUnWinderAxisB.commands.posAbsolute AND ("Unit1.Em0.HmiInterface".cmUnWinderAxisB.commandConfiguration.posAbsolute.velocity > #SpeedLimit);
   IF #_w4 THEN
       "Unit1.Em0.HmiInterface".cmUnWinderAxisB.commandConfiguration.posAbsolute.velocity := #SpeedLimit;
       "Unit1.Em0.ControlNodes".cmUnWinderAxisB.commandConfiguration.posAbsolute.velocity := #SpeedLimit;
   END_IF;
END_REGION

REGION Network 52: Call CM Unwinder B Axis (LBC_AxisControl)
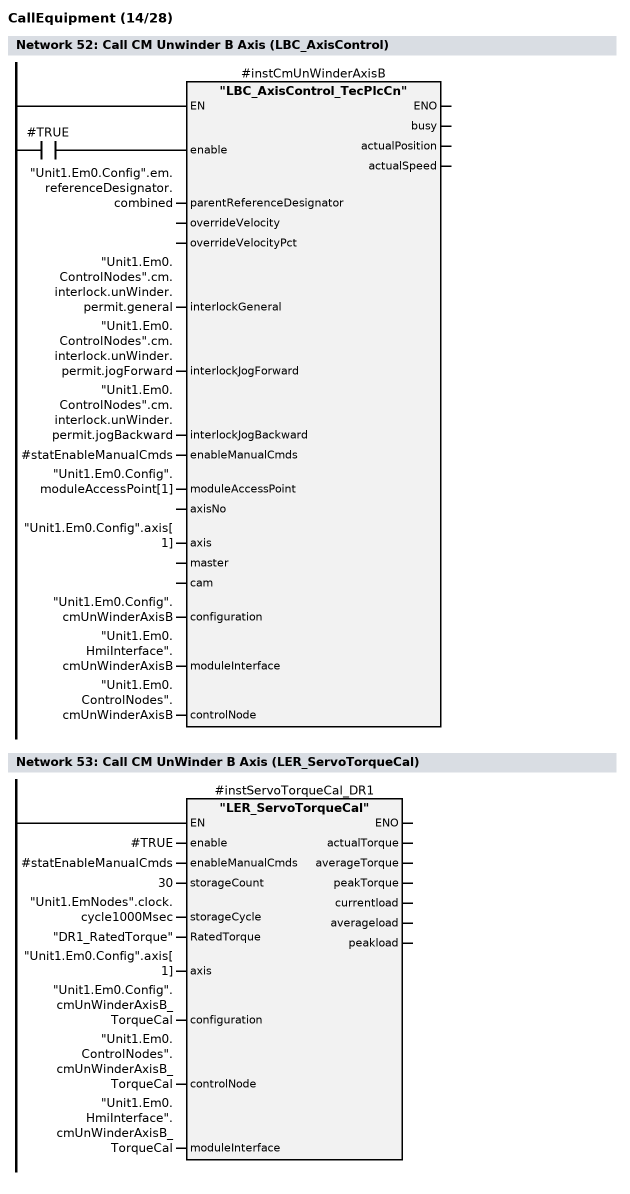
   RUNG wire#powerrail
      #instCmUnWinderAxisB(enable := wire#w1, parentReferenceDesignator := "Unit1.Em0.Config".em.referenceDesignator.combined, overrideVelocity :=, overrideVelocityPct :=, interlockGeneral := "Unit1.Em0.ControlNodes".cm.interlock.unWinder.permit.general, interlockJogForward := "Unit1.Em0.ControlNodes".cm.interlock.unWinder.permit.jogForward, interlockJogBackward := "Unit1.Em0.ControlNodes".cm.interlock.unWinder.permit.jogBackward, enableManualCmds := #statEnableManualCmds, moduleAccessPoint := "Unit1.Em0.Config".moduleAccessPoint[1], axisNo :=, axis := "Unit1.Em0.Config".axis[1], master :=, cam :=, configuration := "Unit1.Em0.Config".cmUnWinderAxisB, moduleInterface := "Unit1.Em0.HmiInterface".cmUnWinderAxisB, controlNode := "Unit1.Em0.ControlNodes".cmUnWinderAxisB, busy =>, actualPosition =>, actualSpeed =>)
   END_RUNG
   RUNG wire#powerrail
      Contact( #TRUE )
   END_RUNG wire#w1
   // the same network as SCL:
   #instCmUnWinderAxisB(enable := #TRUE,   // "LBC_AxisControl_TecPlcCn"
                        parentReferenceDesignator := "Unit1.Em0.Config".em.referenceDesignator.combined,
                        interlockGeneral := "Unit1.Em0.ControlNodes".cm.interlock.unWinder.permit.general,
                        interlockJogForward := "Unit1.Em0.ControlNodes".cm.interlock.unWinder.permit.jogForward,
                        interlockJogBackward := "Unit1.Em0.ControlNodes".cm.interlock.unWinder.permit.jogBackward,
                        enableManualCmds := #statEnableManualCmds,
                        moduleAccessPoint := "Unit1.Em0.Config".moduleAccessPoint[1],
                        axis := "Unit1.Em0.Config".axis[1],
                        configuration := "Unit1.Em0.Config".cmUnWinderAxisB,
                        moduleInterface := "Unit1.Em0.HmiInterface".cmUnWinderAxisB,
                        controlNode := "Unit1.Em0.ControlNodes".cmUnWinderAxisB);
END_REGION

REGION Network 53: Call CM UnWinder B Axis (LER_ServoTorqueCal)
   RUNG wire#powerrail
      #instServoTorqueCal_DR1(enable := #TRUE, enableManualCmds := #statEnableManualCmds, storageCount := 30, storageCycle := "Unit1.EmNodes".clock.cycle1000Msec, RatedTorque := "DR1_RatedTorque", axis := "Unit1.Em0.Config".axis[1], configuration := "Unit1.Em0.Config".cmUnWinderAxisB_TorqueCal, controlNode := "Unit1.Em0.ControlNodes".cmUnWinderAxisB_TorqueCal, moduleInterface := "Unit1.Em0.HmiInterface".cmUnWinderAxisB_TorqueCal, actualTorque =>, averageTorque =>, peakTorque =>, currentload =>, averageload =>, peakload =>)
   END_RUNG
   // the same network as SCL:
   #instServoTorqueCal_DR1(enable := #TRUE,   // "LER_ServoTorqueCal"
                           enableManualCmds := #statEnableManualCmds,
                           storageCount := 30,
                           storageCycle := "Unit1.EmNodes".clock.cycle1000Msec,
                           RatedTorque := "DR1_RatedTorque",
                           axis := "Unit1.Em0.Config".axis[1],
                           configuration := "Unit1.Em0.Config".cmUnWinderAxisB_TorqueCal,
                           controlNode := "Unit1.Em0.ControlNodes".cmUnWinderAxisB_TorqueCal,
                           moduleInterface := "Unit1.Em0.HmiInterface".cmUnWinderAxisB_TorqueCal);
END_REGION

REGION Network 55: ******************** Brake Test (Axis) ********************
END_REGION

REGION Network 56: Unwinder Brake Test Error
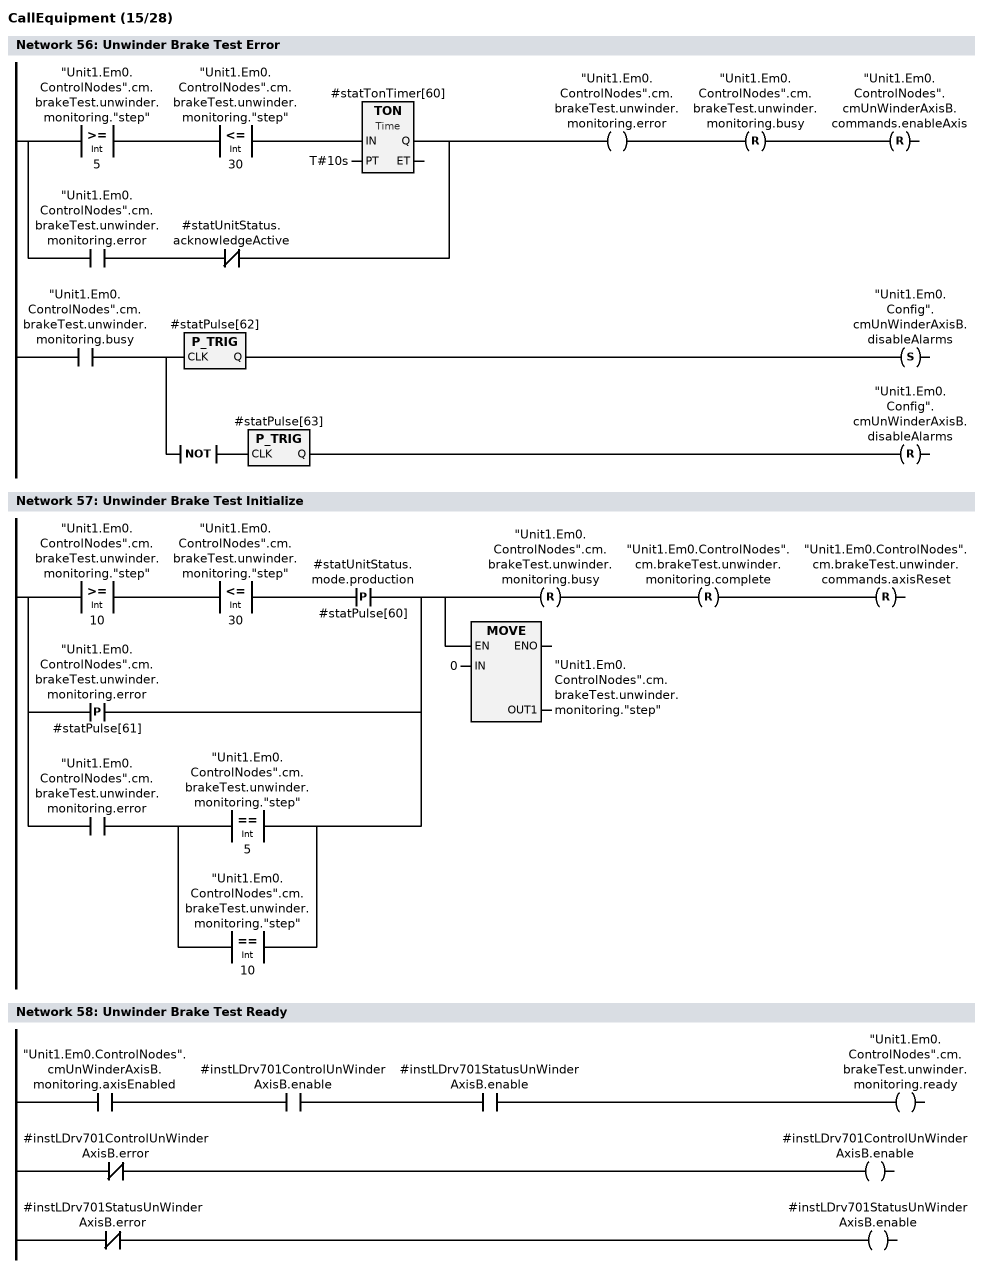
   RUNG wire#powerrail
      { S7_Templates := "SrcType := Int" } GE_Contact(in1 := "Unit1.Em0.ControlNodes".cm.brakeTest.unwinder.monitoring."step", in2 := 5)
      { S7_Templates := "SrcType := Int" } LE_Contact(in1 := "Unit1.Em0.ControlNodes".cm.brakeTest.unwinder.monitoring."step", in2 := 30)
      { S7_Templates := "time_type := Time" } #statTonTimer[60].TON(pt := T#10s, et =>)
      wire#w1
      Coil( "Unit1.Em0.ControlNodes".cm.brakeTest.unwinder.monitoring.error )
      R_Coil( "Unit1.Em0.ControlNodes".cm.brakeTest.unwinder.monitoring.busy )
      R_Coil( "Unit1.Em0.ControlNodes".cmUnWinderAxisB.commands.enableAxis )
   END_RUNG
   RUNG wire#powerrail
      Contact( "Unit1.Em0.ControlNodes".cm.brakeTest.unwinder.monitoring.error )
      I_Contact( #statUnitStatus.acknowledgeActive )
   END_RUNG wire#w1
   RUNG wire#powerrail
      Contact( "Unit1.Em0.ControlNodes".cm.brakeTest.unwinder.monitoring.busy )
      wire#w2
      P_Trig( #statPulse[62] )
      S_Coil( "Unit1.Em0.Config".cmUnWinderAxisB.disableAlarms )
   END_RUNG
   RUNG wire#w2
      Not()
      P_Trig( #statPulse[63] )
      R_Coil( "Unit1.Em0.Config".cmUnWinderAxisB.disableAlarms )
   END_RUNG
   // the same network as SCL:
   #statTonTimer[60].TON(IN := ("Unit1.Em0.ControlNodes".cm.brakeTest.unwinder.monitoring."step" >= 5) AND ("Unit1.Em0.ControlNodes".cm.brakeTest.unwinder.monitoring."step" <= 30),
                         PT := T#10s);
   "Unit1.Em0.ControlNodes".cm.brakeTest.unwinder.monitoring.error := #statTonTimer[60].Q OR ("Unit1.Em0.ControlNodes".cm.brakeTest.unwinder.monitoring.error AND NOT #statUnitStatus.acknowledgeActive);
   IF "Unit1.Em0.ControlNodes".cm.brakeTest.unwinder.monitoring.error THEN
       "Unit1.Em0.ControlNodes".cm.brakeTest.unwinder.monitoring.busy := FALSE;
       "Unit1.Em0.ControlNodes".cmUnWinderAxisB.commands.enableAxis := FALSE;
   END_IF;
   #_w1 := "Unit1.Em0.ControlNodes".cm.brakeTest.unwinder.monitoring.busy AND NOT #statPulse[62];   // rising edge
   #statPulse[62] := "Unit1.Em0.ControlNodes".cm.brakeTest.unwinder.monitoring.busy;
   IF #_w1 THEN "Unit1.Em0.Config".cmUnWinderAxisB.disableAlarms := TRUE; END_IF;
   #_w2 := NOT "Unit1.Em0.ControlNodes".cm.brakeTest.unwinder.monitoring.busy AND NOT #statPulse[63];   // rising edge
   #statPulse[63] := NOT "Unit1.Em0.ControlNodes".cm.brakeTest.unwinder.monitoring.busy;
   IF #_w2 THEN "Unit1.Em0.Config".cmUnWinderAxisB.disableAlarms := FALSE; END_IF;
END_REGION

REGION Network 57: Unwinder Brake Test Initialize
   RUNG wire#powerrail
      { S7_Templates := "SrcType := Int" } GE_Contact(in1 := "Unit1.Em0.ControlNodes".cm.brakeTest.unwinder.monitoring."step", in2 := 10)
      { S7_Templates := "SrcType := Int" } LE_Contact(in1 := "Unit1.Em0.ControlNodes".cm.brakeTest.unwinder.monitoring."step", in2 := 30)
      P_Contact(operand := #statUnitStatus.mode.production, bit := #statPulse[60])
      wire#w1
      R_Coil( "Unit1.Em0.ControlNodes".cm.brakeTest.unwinder.monitoring.busy )
      R_Coil( "Unit1.Em0.ControlNodes".cm.brakeTest.unwinder.monitoring.complete )
      R_Coil( "Unit1.Em0.ControlNodes".cm.brakeTest.unwinder.commands.axisReset )
   END_RUNG
   RUNG wire#powerrail
      P_Contact(operand := "Unit1.Em0.ControlNodes".cm.brakeTest.unwinder.monitoring.error, bit := #statPulse[61])
   END_RUNG wire#w1
   RUNG wire#powerrail
      Contact( "Unit1.Em0.ControlNodes".cm.brakeTest.unwinder.monitoring.error )
      wire#w2
      { S7_Templates := "SrcType := Int" } EQ_Contact(in1 := "Unit1.Em0.ControlNodes".cm.brakeTest.unwinder.monitoring."step", in2 := 5)
   END_RUNG wire#w1
   RUNG wire#w2
      { S7_Templates := "SrcType := Int" } EQ_Contact(in1 := "Unit1.Em0.ControlNodes".cm.brakeTest.unwinder.monitoring."step", in2 := 10)
   END_RUNG wire#w1
   RUNG wire#w1
      Move(in := 0, out1 => "Unit1.Em0.ControlNodes".cm.brakeTest.unwinder.monitoring."step")
   END_RUNG
   // the same network as SCL:
   #_w1 := ("Unit1.Em0.ControlNodes".cm.brakeTest.unwinder.monitoring."step" >= 10) AND ("Unit1.Em0.ControlNodes".cm.brakeTest.unwinder.monitoring."step" <= 30) AND #statUnitStatus.mode.production AND NOT #statPulse[60];   // rising edge of #statUnitStatus.mode.production
   #statPulse[60] := #statUnitStatus.mode.production;
   #_w2 := "Unit1.Em0.ControlNodes".cm.brakeTest.unwinder.monitoring.error AND NOT #statPulse[61];   // rising edge of "Unit1.Em0.ControlNodes".cm.brakeTest.unwinder.monitoring.error
   #statPulse[61] := "Unit1.Em0.ControlNodes".cm.brakeTest.unwinder.monitoring.error;
   IF #_w1 OR #_w2 OR ("Unit1.Em0.ControlNodes".cm.brakeTest.unwinder.monitoring.error AND (("Unit1.Em0.ControlNodes".cm.brakeTest.unwinder.monitoring."step" = 5) OR ("Unit1.Em0.ControlNodes".cm.brakeTest.unwinder.monitoring."step" = 10))) THEN
       "Unit1.Em0.ControlNodes".cm.brakeTest.unwinder.monitoring.busy := FALSE;
       "Unit1.Em0.ControlNodes".cm.brakeTest.unwinder.monitoring.complete := FALSE;
       "Unit1.Em0.ControlNodes".cm.brakeTest.unwinder.commands.axisReset := FALSE;
       "Unit1.Em0.ControlNodes".cm.brakeTest.unwinder.monitoring."step" := 0;
   END_IF;
END_REGION

REGION Network 58: Unwinder Brake Test Ready
   RUNG wire#powerrail
      Contact( "Unit1.Em0.ControlNodes".cmUnWinderAxisB.monitoring.axisEnabled )
      Contact( #instLDrv701ControlUnWinderAxisB.enable )
      Contact( #instLDrv701StatusUnWinderAxisB.enable )
      Coil( "Unit1.Em0.ControlNodes".cm.brakeTest.unwinder.monitoring.ready )
   END_RUNG
   RUNG wire#powerrail
      I_Contact( #instLDrv701ControlUnWinderAxisB.error )
      Coil( #instLDrv701ControlUnWinderAxisB.enable )
   END_RUNG
   RUNG wire#powerrail
      I_Contact( #instLDrv701StatusUnWinderAxisB.error )
      Coil( #instLDrv701StatusUnWinderAxisB.enable )
   END_RUNG
   // the same network as SCL:
   "Unit1.Em0.ControlNodes".cm.brakeTest.unwinder.monitoring.ready := "Unit1.Em0.ControlNodes".cmUnWinderAxisB.monitoring.axisEnabled AND #instLDrv701ControlUnWinderAxisB.enable AND #instLDrv701StatusUnWinderAxisB.enable;
   #instLDrv701ControlUnWinderAxisB.enable := NOT #instLDrv701ControlUnWinderAxisB.error;
   #instLDrv701StatusUnWinderAxisB.enable := NOT #instLDrv701StatusUnWinderAxisB.error;
END_REGION

REGION Network 59: Unwinder Axis Reset
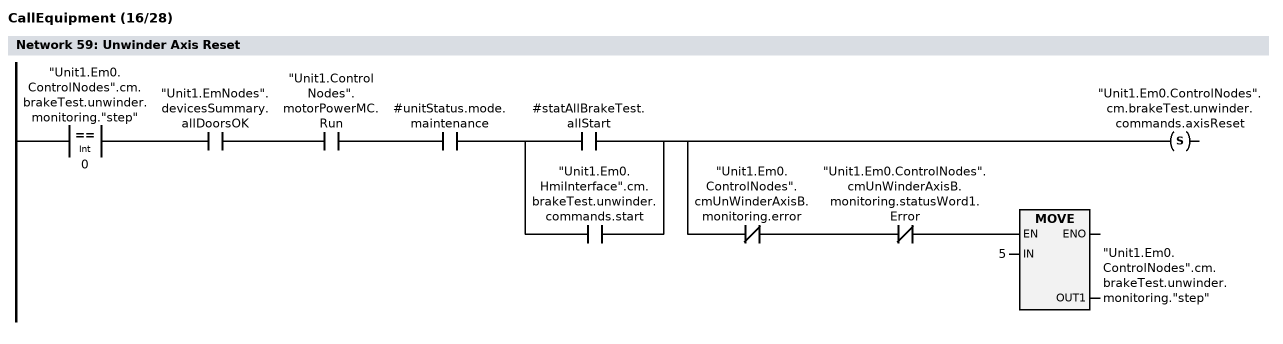
   RUNG wire#powerrail
      { S7_Templates := "SrcType := Int" } EQ_Contact(in1 := "Unit1.Em0.ControlNodes".cm.brakeTest.unwinder.monitoring."step", in2 := 0)
      Contact( "Unit1.EmNodes".devicesSummary.allDoorsOK )
      Contact( "Unit1.ControlNodes".motorPowerMC.Run )
      Contact( #unitStatus.mode.maintenance )
      wire#w1
      Contact( #statAllBrakeTest.allStart )
      wire#w2
      S_Coil( "Unit1.Em0.ControlNodes".cm.brakeTest.unwinder.commands.axisReset )
   END_RUNG
   RUNG wire#w1
      Contact( "Unit1.Em0.HmiInterface".cm.brakeTest.unwinder.commands.start )
   END_RUNG wire#w2
   RUNG wire#w2
      I_Contact( "Unit1.Em0.ControlNodes".cmUnWinderAxisB.monitoring.error )
      I_Contact( "Unit1.Em0.ControlNodes".cmUnWinderAxisB.monitoring.statusWord1.Error )
      Move(in := 5, out1 => "Unit1.Em0.ControlNodes".cm.brakeTest.unwinder.monitoring."step")
   END_RUNG
   // the same network as SCL:
   #_w1 := ("Unit1.Em0.ControlNodes".cm.brakeTest.unwinder.monitoring."step" = 0) AND "Unit1.EmNodes".devicesSummary.allDoorsOK AND "Unit1.ControlNodes".motorPowerMC.Run AND #unitStatus.mode.maintenance AND (#statAllBrakeTest.allStart OR "Unit1.Em0.HmiInterface".cm.brakeTest.unwinder.commands.start);
   IF #_w1 THEN "Unit1.Em0.ControlNodes".cm.brakeTest.unwinder.commands.axisReset := TRUE; END_IF;
   IF #_w1 AND NOT "Unit1.Em0.ControlNodes".cmUnWinderAxisB.monitoring.error AND NOT "Unit1.Em0.ControlNodes".cmUnWinderAxisB.monitoring.statusWord1.Error THEN
       "Unit1.Em0.ControlNodes".cm.brakeTest.unwinder.monitoring."step" := 5;
   END_IF;
END_REGION

REGION Network 60: Unwinder Brake Test Commands
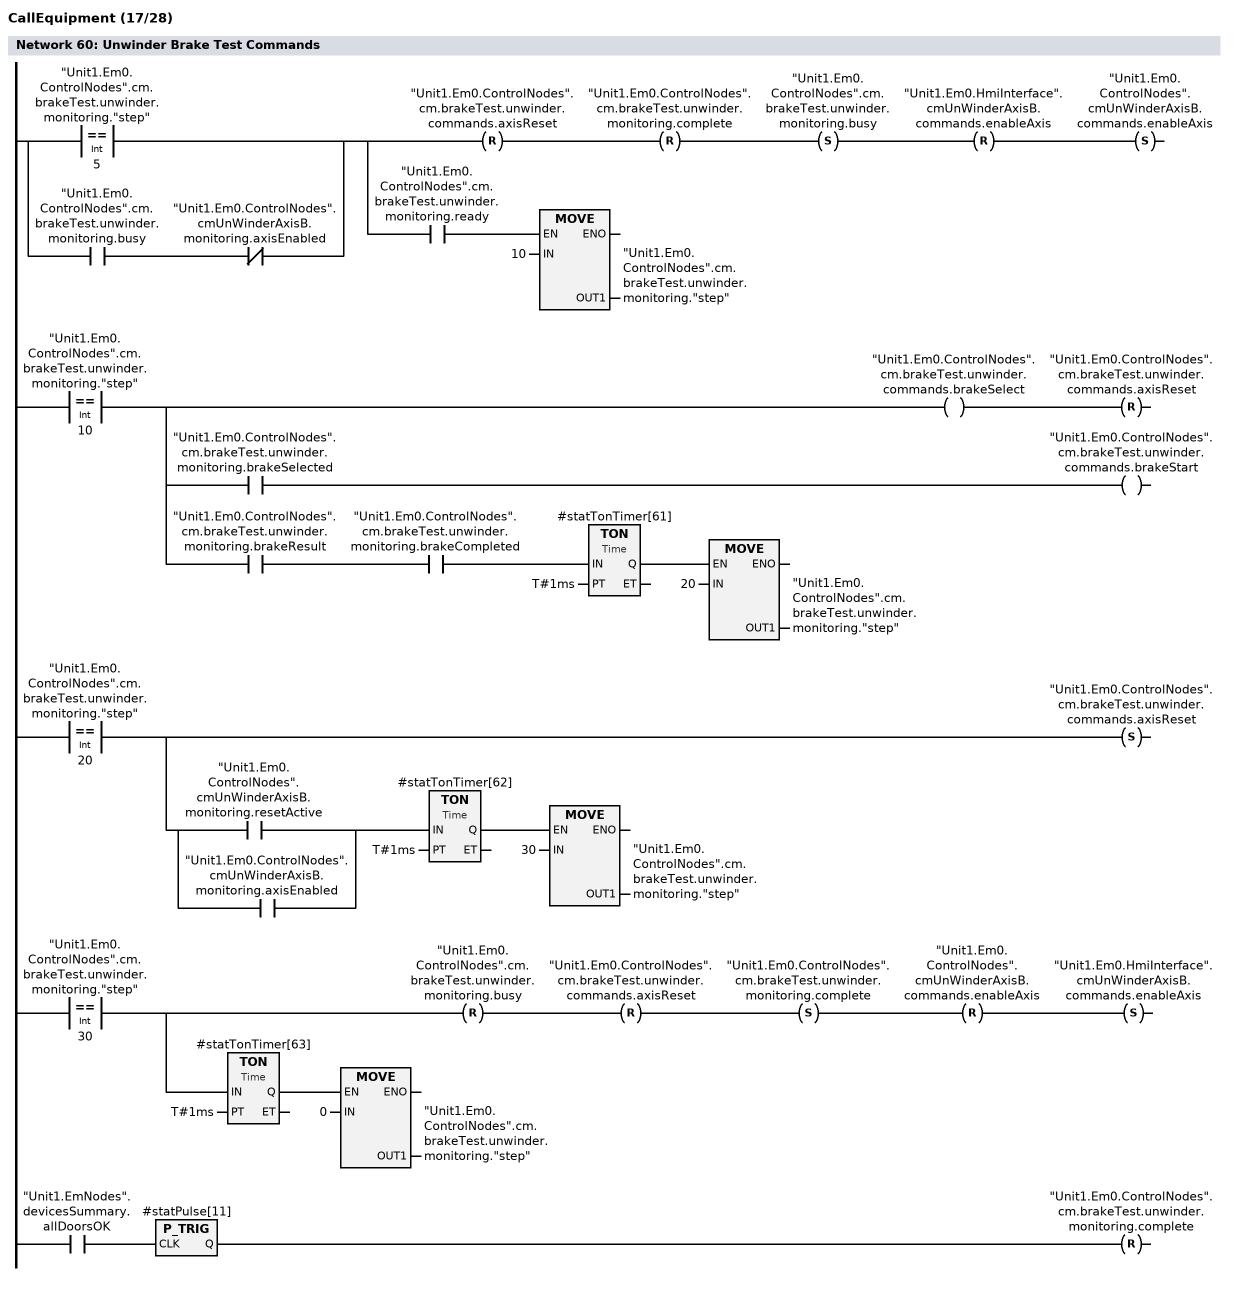
   RUNG wire#powerrail
      { S7_Templates := "SrcType := Int" } EQ_Contact(in1 := "Unit1.Em0.ControlNodes".cm.brakeTest.unwinder.monitoring."step", in2 := 5)
      wire#w1
      R_Coil( "Unit1.Em0.ControlNodes".cm.brakeTest.unwinder.commands.axisReset )
      R_Coil( "Unit1.Em0.ControlNodes".cm.brakeTest.unwinder.monitoring.complete )
      S_Coil( "Unit1.Em0.ControlNodes".cm.brakeTest.unwinder.monitoring.busy )
      R_Coil( "Unit1.Em0.HmiInterface".cmUnWinderAxisB.commands.enableAxis )
      S_Coil( "Unit1.Em0.ControlNodes".cmUnWinderAxisB.commands.enableAxis )
   END_RUNG
   RUNG wire#powerrail
      Contact( "Unit1.Em0.ControlNodes".cm.brakeTest.unwinder.monitoring.busy )
      I_Contact( "Unit1.Em0.ControlNodes".cmUnWinderAxisB.monitoring.axisEnabled )
   END_RUNG wire#w1
   RUNG wire#w1
      Contact( "Unit1.Em0.ControlNodes".cm.brakeTest.unwinder.monitoring.ready )
      Move(in := 10, out1 => "Unit1.Em0.ControlNodes".cm.brakeTest.unwinder.monitoring."step")
   END_RUNG
   RUNG wire#powerrail
      { S7_Templates := "SrcType := Int" } EQ_Contact(in1 := "Unit1.Em0.ControlNodes".cm.brakeTest.unwinder.monitoring."step", in2 := 10)
      wire#w2
      Coil( "Unit1.Em0.ControlNodes".cm.brakeTest.unwinder.commands.brakeSelect )
      R_Coil( "Unit1.Em0.ControlNodes".cm.brakeTest.unwinder.commands.axisReset )
   END_RUNG
   RUNG wire#w2
      Contact( "Unit1.Em0.ControlNodes".cm.brakeTest.unwinder.monitoring.brakeSelected )
      Coil( "Unit1.Em0.ControlNodes".cm.brakeTest.unwinder.commands.brakeStart )
   END_RUNG
   RUNG wire#w2
      Contact( "Unit1.Em0.ControlNodes".cm.brakeTest.unwinder.monitoring.brakeResult )
      Contact( "Unit1.Em0.ControlNodes".cm.brakeTest.unwinder.monitoring.brakeCompleted )
      { S7_Templates := "time_type := Time" } #statTonTimer[61].TON(pt := T#1ms, et =>)
      Move(in := 20, out1 => "Unit1.Em0.ControlNodes".cm.brakeTest.unwinder.monitoring."step")
   END_RUNG
   RUNG wire#powerrail
      { S7_Templates := "SrcType := Int" } EQ_Contact(in1 := "Unit1.Em0.ControlNodes".cm.brakeTest.unwinder.monitoring."step", in2 := 20)
      wire#w3
      S_Coil( "Unit1.Em0.ControlNodes".cm.brakeTest.unwinder.commands.axisReset )
   END_RUNG
   RUNG wire#w3
      Contact( "Unit1.Em0.ControlNodes".cmUnWinderAxisB.monitoring.resetActive )
      wire#w4
      { S7_Templates := "time_type := Time" } #statTonTimer[62].TON(pt := T#1ms, et =>)
      Move(in := 30, out1 => "Unit1.Em0.ControlNodes".cm.brakeTest.unwinder.monitoring."step")
   END_RUNG
   RUNG wire#w3
      Contact( "Unit1.Em0.ControlNodes".cmUnWinderAxisB.monitoring.axisEnabled )
   END_RUNG wire#w4
   RUNG wire#powerrail
      { S7_Templates := "SrcType := Int" } EQ_Contact(in1 := "Unit1.Em0.ControlNodes".cm.brakeTest.unwinder.monitoring."step", in2 := 30)
      wire#w5
      R_Coil( "Unit1.Em0.ControlNodes".cm.brakeTest.unwinder.monitoring.busy )
      R_Coil( "Unit1.Em0.ControlNodes".cm.brakeTest.unwinder.commands.axisReset )
      S_Coil( "Unit1.Em0.ControlNodes".cm.brakeTest.unwinder.monitoring.complete )
      R_Coil( "Unit1.Em0.ControlNodes".cmUnWinderAxisB.commands.enableAxis )
      S_Coil( "Unit1.Em0.HmiInterface".cmUnWinderAxisB.commands.enableAxis )
   END_RUNG
   RUNG wire#w5
      { S7_Templates := "time_type := Time" } #statTonTimer[63].TON(pt := T#1ms, et =>)
      Move(in := 0, out1 => "Unit1.Em0.ControlNodes".cm.brakeTest.unwinder.monitoring."step")
   END_RUNG
   RUNG wire#powerrail
      Contact( "Unit1.EmNodes".devicesSummary.allDoorsOK )
      P_Trig( #statPulse[11] )
      R_Coil( "Unit1.Em0.ControlNodes".cm.brakeTest.unwinder.monitoring.complete )
   END_RUNG
   // the same network as SCL:
   #_w1 := ("Unit1.Em0.ControlNodes".cm.brakeTest.unwinder.monitoring."step" = 5) OR ("Unit1.Em0.ControlNodes".cm.brakeTest.unwinder.monitoring.busy AND NOT "Unit1.Em0.ControlNodes".cmUnWinderAxisB.monitoring.axisEnabled);
   IF #_w1 THEN
       "Unit1.Em0.ControlNodes".cm.brakeTest.unwinder.commands.axisReset := FALSE;
       "Unit1.Em0.ControlNodes".cm.brakeTest.unwinder.monitoring.complete := FALSE;
       "Unit1.Em0.ControlNodes".cm.brakeTest.unwinder.monitoring.busy := TRUE;
       "Unit1.Em0.HmiInterface".cmUnWinderAxisB.commands.enableAxis := FALSE;
       "Unit1.Em0.ControlNodes".cmUnWinderAxisB.commands.enableAxis := TRUE;
   END_IF;
   IF #_w1 AND "Unit1.Em0.ControlNodes".cm.brakeTest.unwinder.monitoring.ready THEN
       "Unit1.Em0.ControlNodes".cm.brakeTest.unwinder.monitoring."step" := 10;
   END_IF;
   "Unit1.Em0.ControlNodes".cm.brakeTest.unwinder.commands.brakeSelect := "Unit1.Em0.ControlNodes".cm.brakeTest.unwinder.monitoring."step" = 10;
   IF "Unit1.Em0.ControlNodes".cm.brakeTest.unwinder.commands.brakeSelect THEN
       "Unit1.Em0.ControlNodes".cm.brakeTest.unwinder.commands.axisReset := FALSE;
   END_IF;
   "Unit1.Em0.ControlNodes".cm.brakeTest.unwinder.commands.brakeStart := "Unit1.Em0.ControlNodes".cm.brakeTest.unwinder.commands.brakeSelect AND "Unit1.Em0.ControlNodes".cm.brakeTest.unwinder.monitoring.brakeSelected;
   #statTonTimer[61].TON(IN := "Unit1.Em0.ControlNodes".cm.brakeTest.unwinder.commands.brakeSelect AND "Unit1.Em0.ControlNodes".cm.brakeTest.unwinder.monitoring.brakeResult AND "Unit1.Em0.ControlNodes".cm.brakeTest.unwinder.monitoring.brakeCompleted,
                         PT := T#1ms);
   IF #statTonTimer[61].Q THEN
       "Unit1.Em0.ControlNodes".cm.brakeTest.unwinder.monitoring."step" := 20;
   END_IF;
   #_w2 := "Unit1.Em0.ControlNodes".cm.brakeTest.unwinder.monitoring."step" = 20;
   IF #_w2 THEN "Unit1.Em0.ControlNodes".cm.brakeTest.unwinder.commands.axisReset := TRUE; END_IF;
   #statTonTimer[62].TON(IN := #_w2 AND ("Unit1.Em0.ControlNodes".cmUnWinderAxisB.monitoring.resetActive OR "Unit1.Em0.ControlNodes".cmUnWinderAxisB.monitoring.axisEnabled),
                         PT := T#1ms);
   IF #statTonTimer[62].Q THEN
       "Unit1.Em0.ControlNodes".cm.brakeTest.unwinder.monitoring."step" := 30;
   END_IF;
   #_w3 := "Unit1.Em0.ControlNodes".cm.brakeTest.unwinder.monitoring."step" = 30;
   IF #_w3 THEN
       "Unit1.Em0.ControlNodes".cm.brakeTest.unwinder.monitoring.busy := FALSE;
       "Unit1.Em0.ControlNodes".cm.brakeTest.unwinder.commands.axisReset := FALSE;
       "Unit1.Em0.ControlNodes".cm.brakeTest.unwinder.monitoring.complete := TRUE;
       "Unit1.Em0.ControlNodes".cmUnWinderAxisB.commands.enableAxis := FALSE;
       "Unit1.Em0.HmiInterface".cmUnWinderAxisB.commands.enableAxis := TRUE;
   END_IF;
   #statTonTimer[63].TON(IN := #_w3, PT := T#1ms);
   IF #statTonTimer[63].Q THEN "Unit1.Em0.ControlNodes".cm.brakeTest.unwinder.monitoring."step" := 0; END_IF;
   #_w4 := "Unit1.EmNodes".devicesSummary.allDoorsOK AND NOT #statPulse[11];   // rising edge
   #statPulse[11] := "Unit1.EmNodes".devicesSummary.allDoorsOK;
   IF #_w4 THEN "Unit1.Em0.ControlNodes".cm.brakeTest.unwinder.monitoring.complete := FALSE; END_IF;
END_REGION

REGION Network 61: Unwinder Brake Test Monitoring
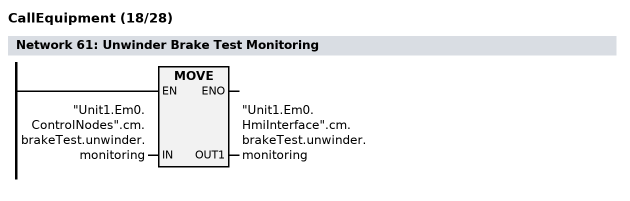
   RUNG wire#powerrail
      Move(in := "Unit1.Em0.ControlNodes".cm.brakeTest.unwinder.monitoring, out1 => "Unit1.Em0.HmiInterface".cm.brakeTest.unwinder.monitoring)
   END_RUNG
   // the same network as SCL:
   "Unit1.Em0.HmiInterface".cm.brakeTest.unwinder.monitoring := "Unit1.Em0.ControlNodes".cm.brakeTest.unwinder.monitoring;
END_REGION

REGION Network 62: Unwinder Telegram 701
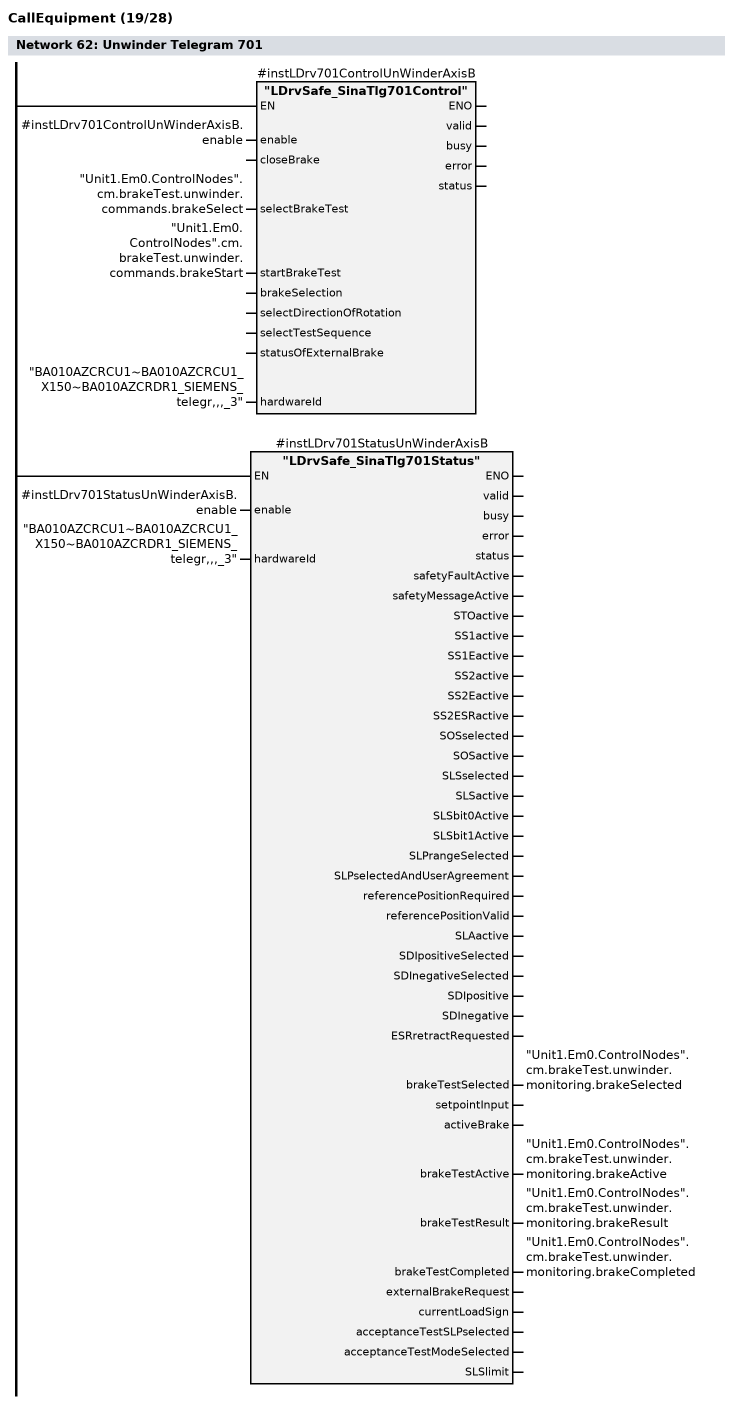
   RUNG wire#powerrail
      #instLDrv701ControlUnWinderAxisB(enable := #instLDrv701ControlUnWinderAxisB.enable, closeBrake :=, selectBrakeTest := "Unit1.Em0.ControlNodes".cm.brakeTest.unwinder.commands.brakeSelect, startBrakeTest := "Unit1.Em0.ControlNodes".cm.brakeTest.unwinder.commands.brakeStart, brakeSelection :=, selectDirectionOfRotation :=, selectTestSequence :=, statusOfExternalBrake :=, hardwareId := "BA010AZCRCU1~BA010AZCRCU1_X150~BA010AZCRDR1_SIEMENS_telegr,,,_3", valid =>, busy =>, error =>, status =>)
   END_RUNG
   RUNG wire#powerrail
      #instLDrv701StatusUnWinderAxisB(enable := #instLDrv701StatusUnWinderAxisB.enable, hardwareId := "BA010AZCRCU1~BA010AZCRCU1_X150~BA010AZCRDR1_SIEMENS_telegr,,,_3", valid =>, busy =>, error =>, status =>, safetyFaultActive =>, safetyMessageActive =>, STOactive =>, SS1active =>, SS1Eactive =>, SS2active =>, SS2Eactive =>, SS2ESRactive =>, SOSselected =>, SOSactive =>, SLSselected =>, SLSactive =>, SLSbit0Active =>, SLSbit1Active =>, SLPrangeSelected =>, SLPselectedAndUserAgreement =>, referencePositionRequired =>, referencePositionValid =>, SLAactive =>, SDIpositiveSelected =>, SDInegativeSelected =>, SDIpositive =>, SDInegative =>, ESRretractRequested =>, brakeTestSelected => "Unit1.Em0.ControlNodes".cm.brakeTest.unwinder.monitoring.brakeSelected, setpointInput =>, activeBrake =>, brakeTestActive => "Unit1.Em0.ControlNodes".cm.brakeTest.unwinder.monitoring.brakeActive, brakeTestResult => "Unit1.Em0.ControlNodes".cm.brakeTest.unwinder.monitoring.brakeResult, brakeTestCompleted => "Unit1.Em0.ControlNodes".cm.brakeTest.unwinder.monitoring.brakeCompleted, externalBrakeRequest =>, currentLoadSign =>, acceptanceTestSLPselected =>, acceptanceTestModeSelected =>, SLSlimit =>)
   END_RUNG
   // the same network as SCL:
   #instLDrv701ControlUnWinderAxisB(enable := #instLDrv701ControlUnWinderAxisB.enable,   // "LDrvSafe_SinaTlg701Control"
                           selectBrakeTest := "Unit1.Em0.ControlNodes".cm.brakeTest.unwinder.commands.brakeSelect,
                           startBrakeTest := "Unit1.Em0.ControlNodes".cm.brakeTest.unwinder.commands.brakeStart,
                           hardwareId := "BA010AZCRCU1~BA010AZCRCU1_X150~BA010AZCRDR1_SIEMENS_telegr,,,_3");
   #instLDrv701StatusUnWinderAxisB(enable := #instLDrv701StatusUnWinderAxisB.enable,   // "LDrvSafe_SinaTlg701Status"
                           hardwareId := "BA010AZCRCU1~BA010AZCRCU1_X150~BA010AZCRDR1_SIEMENS_telegr,,,_3",
                           brakeTestSelected => "Unit1.Em0.ControlNodes".cm.brakeTest.unwinder.monitoring.brakeSelected,
                           brakeTestActive => "Unit1.Em0.ControlNodes".cm.brakeTest.unwinder.monitoring.brakeActive,
                           brakeTestResult => "Unit1.Em0.ControlNodes".cm.brakeTest.unwinder.monitoring.brakeResult,
                           brakeTestCompleted => "Unit1.Em0.ControlNodes".cm.brakeTest.unwinder.monitoring.brakeCompleted);
END_REGION

REGION Network 64: ******************** Control Modules (TwoWayActuator) ********************
   // Call control modules that are actuators after the em logic (jobs and sequence), so that the latest commands are applied to the actuators.
END_REGION

REGION Network 65: Reset CMS
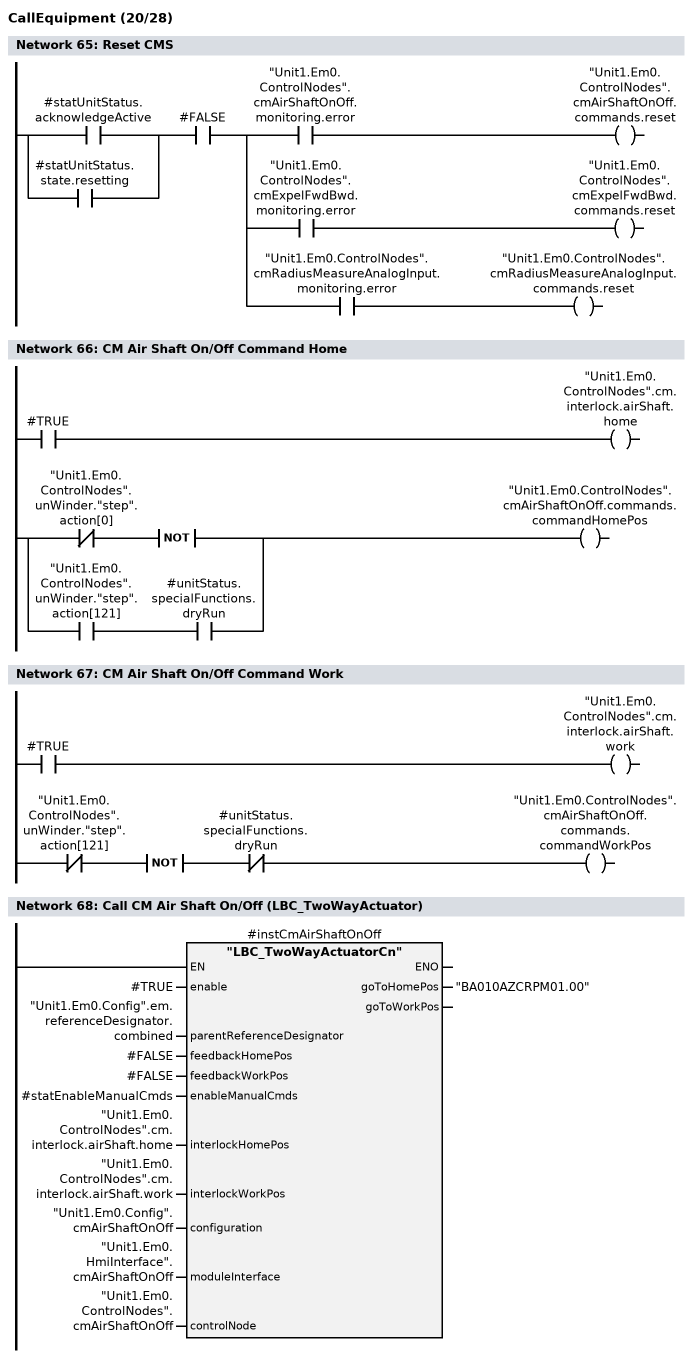
   RUNG wire#powerrail
      Contact( #statUnitStatus.acknowledgeActive )
      wire#w1
      Contact( #FALSE )
      wire#w2
      Contact( "Unit1.Em0.ControlNodes".cmAirShaftOnOff.monitoring.error )
      Coil( "Unit1.Em0.ControlNodes".cmAirShaftOnOff.commands.reset )
   END_RUNG
   RUNG wire#powerrail
      Contact( #statUnitStatus.state.resetting )
   END_RUNG wire#w1
   RUNG wire#w2
      Contact( "Unit1.Em0.ControlNodes".cmExpelFwdBwd.monitoring.error )
      Coil( "Unit1.Em0.ControlNodes".cmExpelFwdBwd.commands.reset )
   END_RUNG
   RUNG wire#w2
      Contact( "Unit1.Em0.ControlNodes".cmRadiusMeasureAnalogInput.monitoring.error )
      Coil( "Unit1.Em0.ControlNodes".cmRadiusMeasureAnalogInput.commands.reset )
   END_RUNG
   // the same network as SCL:
   #_w1 := (#statUnitStatus.acknowledgeActive OR #statUnitStatus.state.resetting) AND #FALSE;
   "Unit1.Em0.ControlNodes".cmAirShaftOnOff.commands.reset := #_w1 AND "Unit1.Em0.ControlNodes".cmAirShaftOnOff.monitoring.error;
   "Unit1.Em0.ControlNodes".cmExpelFwdBwd.commands.reset := #_w1 AND "Unit1.Em0.ControlNodes".cmExpelFwdBwd.monitoring.error;
   "Unit1.Em0.ControlNodes".cmRadiusMeasureAnalogInput.commands.reset := #_w1 AND "Unit1.Em0.ControlNodes".cmRadiusMeasureAnalogInput.monitoring.error;
END_REGION

REGION Network 66: CM Air Shaft On/Off Command Home
   RUNG wire#powerrail
      Contact( #TRUE )
      Coil( "Unit1.Em0.ControlNodes".cm.interlock.airShaft.home )
   END_RUNG
   RUNG wire#powerrail
      I_Contact( "Unit1.Em0.ControlNodes".unWinder."step".action[0] )
      Not()
      wire#w1
      Coil( "Unit1.Em0.ControlNodes".cmAirShaftOnOff.commands.commandHomePos )
   END_RUNG
   RUNG wire#powerrail
      Contact( "Unit1.Em0.ControlNodes".unWinder."step".action[121] )
      Contact( #unitStatus.specialFunctions.dryRun )
   END_RUNG wire#w1
   // the same network as SCL:
   "Unit1.Em0.ControlNodes".cm.interlock.airShaft.home := #TRUE;
   "Unit1.Em0.ControlNodes".cmAirShaftOnOff.commands.commandHomePos := NOT (NOT "Unit1.Em0.ControlNodes".unWinder."step".action[0]) OR ("Unit1.Em0.ControlNodes".unWinder."step".action[121] AND #unitStatus.specialFunctions.dryRun);
END_REGION

REGION Network 67: CM Air Shaft On/Off Command Work
   RUNG wire#powerrail
      Contact( #TRUE )
      Coil( "Unit1.Em0.ControlNodes".cm.interlock.airShaft.work )
   END_RUNG
   RUNG wire#powerrail
      I_Contact( "Unit1.Em0.ControlNodes".unWinder."step".action[121] )
      Not()
      I_Contact( #unitStatus.specialFunctions.dryRun )
      Coil( "Unit1.Em0.ControlNodes".cmAirShaftOnOff.commands.commandWorkPos )
   END_RUNG
   // the same network as SCL:
   "Unit1.Em0.ControlNodes".cm.interlock.airShaft.work := #TRUE;
   "Unit1.Em0.ControlNodes".cmAirShaftOnOff.commands.commandWorkPos := NOT (NOT "Unit1.Em0.ControlNodes".unWinder."step".action[121]) AND NOT #unitStatus.specialFunctions.dryRun;
END_REGION

REGION Network 68: Call CM Air Shaft On/Off (LBC_TwoWayActuator)
   RUNG wire#powerrail
      #instCmAirShaftOnOff(enable := #TRUE, parentReferenceDesignator := "Unit1.Em0.Config".em.referenceDesignator.combined, feedbackHomePos := #FALSE, feedbackWorkPos := #FALSE, enableManualCmds := #statEnableManualCmds, interlockHomePos := "Unit1.Em0.ControlNodes".cm.interlock.airShaft.home, interlockWorkPos := "Unit1.Em0.ControlNodes".cm.interlock.airShaft.work, configuration := "Unit1.Em0.Config".cmAirShaftOnOff, moduleInterface := "Unit1.Em0.HmiInterface".cmAirShaftOnOff, controlNode := "Unit1.Em0.ControlNodes".cmAirShaftOnOff, goToHomePos => "BA010AZCRPM01.00", goToWorkPos =>)
   END_RUNG
   // the same network as SCL:
   #instCmAirShaftOnOff(enable := #TRUE,   // "LBC_TwoWayActuatorCn"
                        parentReferenceDesignator := "Unit1.Em0.Config".em.referenceDesignator.combined,
                        feedbackHomePos := #FALSE,
                        feedbackWorkPos := #FALSE,
                        enableManualCmds := #statEnableManualCmds,
                        interlockHomePos := "Unit1.Em0.ControlNodes".cm.interlock.airShaft.home,
                        interlockWorkPos := "Unit1.Em0.ControlNodes".cm.interlock.airShaft.work,
                        configuration := "Unit1.Em0.Config".cmAirShaftOnOff,
                        moduleInterface := "Unit1.Em0.HmiInterface".cmAirShaftOnOff,
                        controlNode := "Unit1.Em0.ControlNodes".cmAirShaftOnOff,
                        goToHomePos => "BA010AZCRPM01.00");
END_REGION

REGION Network 69: CM Expel FWD/BWD Command Home
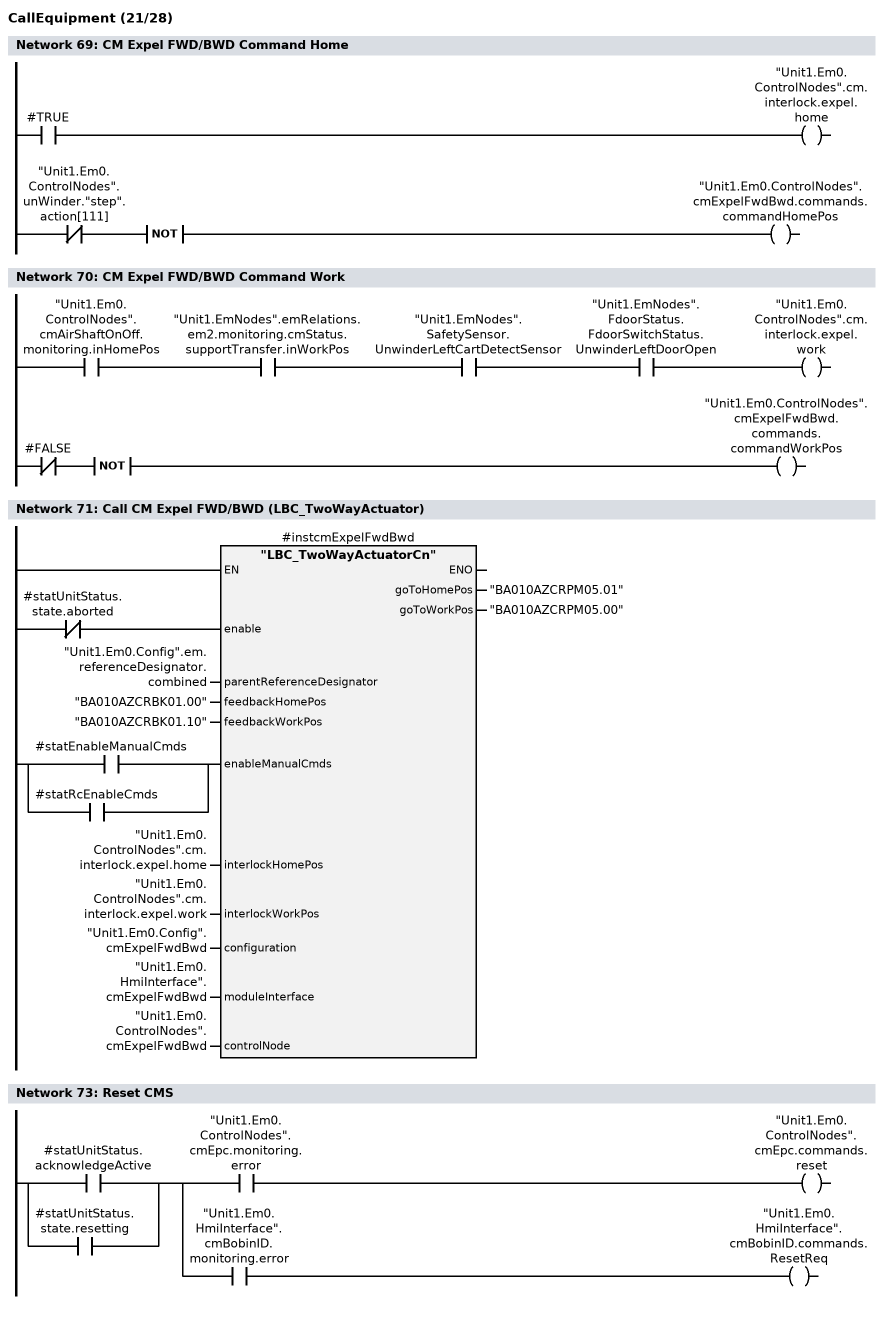
   RUNG wire#powerrail
      Contact( #TRUE )
      Coil( "Unit1.Em0.ControlNodes".cm.interlock.expel.home )
   END_RUNG
   RUNG wire#powerrail
      I_Contact( "Unit1.Em0.ControlNodes".unWinder."step".action[111] )
      Not()
      Coil( "Unit1.Em0.ControlNodes".cmExpelFwdBwd.commands.commandHomePos )
   END_RUNG
   // the same network as SCL:
   "Unit1.Em0.ControlNodes".cm.interlock.expel.home := #TRUE;
   "Unit1.Em0.ControlNodes".cmExpelFwdBwd.commands.commandHomePos := NOT (NOT "Unit1.Em0.ControlNodes".unWinder."step".action[111]);
END_REGION

REGION Network 70: CM Expel FWD/BWD Command Work
   RUNG wire#powerrail
      Contact( "Unit1.Em0.ControlNodes".cmAirShaftOnOff.monitoring.inHomePos )
      Contact( "Unit1.EmNodes".emRelations.em2.monitoring.cmStatus.supportTransfer.inWorkPos )
      Contact( "Unit1.EmNodes".SafetySensor.UnwinderLeftCartDetectSensor )
      Contact( "Unit1.EmNodes".FdoorStatus.FdoorSwitchStatus.UnwinderLeftDoorOpen )
      Coil( "Unit1.Em0.ControlNodes".cm.interlock.expel.work )
   END_RUNG
   RUNG wire#powerrail
      I_Contact( #FALSE )
      Not()
      Coil( "Unit1.Em0.ControlNodes".cmExpelFwdBwd.commands.commandWorkPos )
   END_RUNG
   // the same network as SCL:
   "Unit1.Em0.ControlNodes".cm.interlock.expel.work := "Unit1.Em0.ControlNodes".cmAirShaftOnOff.monitoring.inHomePos AND "Unit1.EmNodes".emRelations.em2.monitoring.cmStatus.supportTransfer.inWorkPos AND "Unit1.EmNodes".SafetySensor.UnwinderLeftCartDetectSensor AND "Unit1.EmNodes".FdoorStatus.FdoorSwitchStatus.UnwinderLeftDoorOpen;
   "Unit1.Em0.ControlNodes".cmExpelFwdBwd.commands.commandWorkPos := NOT (NOT #FALSE);
END_REGION

